KUKA KRL program: MyProgram_285().src

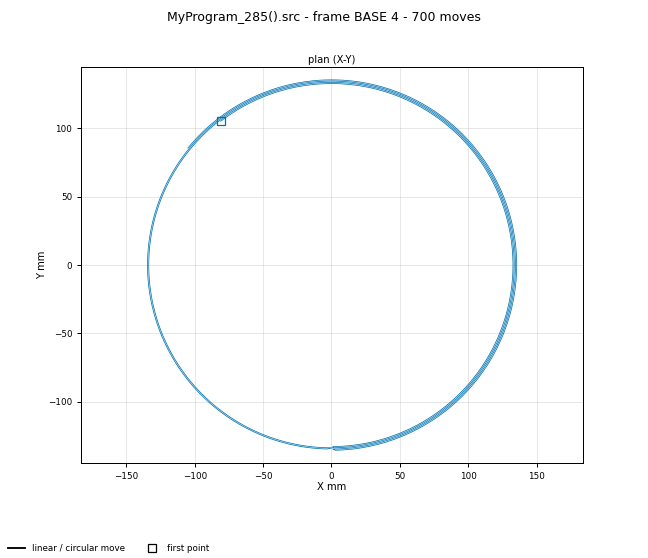
[picture p0: tool path of MyProgram_285().src in frame BASE 4, 700 of 700 moves have a stored position in this frame; points joined in program order, loops and branches not executed]
&ACCESS RVP
&REL 1
&PARAM TEMPLATE = C:\KRC\Roboter\Template\vorgabe
&PARAM EDITMASK = *
DEF MyProgram_285()
; ---- Setting reference (Base) ----
$BASE = BASE_DATA[4]

; --------------------------
; ---- Setting tool (TCP) ----
$TOOL = TOOL_DATA[3]
; --------------------------

$VEL.CP = VEL_APROX_PRINT
Startdeposition()
$VEL.CP = VEL_PRINT
LIN {X -81.057,Y 105.1926,Z 175,A 128.0118,B 7.901,C 0.1192,E1 7.8061,E2 323.7668} C_DIS
LIN {X -78.056,Y 107.4376,Z 175,A 126.422,B 7.9011,C 0.116,E1 7.8097,E2 325.352} C_DIS
LIN {X -74.6273,Y 109.8471,Z 175,A 124.5253,B 7.9011,C 0.1143,E1 7.8141,E2 327.2575} C_DIS
LIN {X -71.0281,Y 112.2079,Z 175,A 122.8509,B 7.9012,C 0.1087,E1 7.818,E2 328.9089} C_DIS
LIN {X -68.5302,Y 113.7507,Z 175,A 121.4995,B 7.9012,C 0.108,E1 7.8212,E2 330.2692} C_DIS
LIN {X -65.7271,Y 115.3929,Z 175,A 120.0866,B 7.9012,C 0.1062,E1 7.8246,E2 331.6823} C_DIS
LIN {X -62.604,Y 117.117,Z 175,A 118.509,B 7.9012,C 0.1046,E1 7.8285,E2 333.2631} C_DIS
LIN {X -59.7165,Y 118.6142,Z 175,A 117.111,B 7.9013,C 0.1027,E1 7.832,E2 334.6594} C_DIS
LIN {X -57.0613,Y 119.9128,Z 175,A 115.7895,B 7.9013,C 0.1017,E1 7.8353,E2 335.9852} C_DIS
LIN {X -53.8159,Y 121.4046,Z 175,A 114.2757,B 7.9013,C 0.0995,E1 7.8391,E2 337.4947} C_DIS
LIN {X -50.7871,Y 122.7025,Z 175,A 112.8825,B 7.9013,C 0.0974,E1 7.8427,E2 338.8834} C_DIS
LIN {X -48.0628,Y 123.7943,Z 175,A 111.5238,B 7.9013,C 0.0974,E1 7.8463,E2 340.252} C_DIS
LIN {X -44.7285,Y 125.0381,Z 175,A 110.0261,B 7.9013,C 0.0954,E1 7.8502,E2 341.7442} C_DIS
LIN {X -41.9571,Y 125.9947,Z 175,A 108.7023,B 7.9013,C 0.0951,E1 7.8537,E2 343.0739} C_DIS
LIN {X -38.5596,Y 127.0761,Z 175,A 107.2508,B 7.9014,C 0.0924,E1 7.8575,E2 344.5142} C_DIS
LIN {X -35.4154,Y 127.9882,Z 175,A 105.7886,B 7.9014,C 0.0921,E1 7.8615,E2 345.9813} C_DIS
LIN {X -32.266,Y 128.8183,Z 175,A 104.3779,B 7.9014,C 0.0911,E1 7.8653,E2 347.3918} C_DIS
LIN {X -29.4073,Y 129.5003,Z 175,A 103.0632,B 7.9014,C 0.0911,E1 7.8689,E2 348.711} C_DIS
LIN {X -25.8996,Y 130.2485,Z 175,A 101.5728,B 7.9014,C 0.0892,E1 7.873,E2 350.1939} C_DIS
LIN {X -22.6971,Y 130.8452,Z 175,A 100.1492,B 7.9014,C 0.0888,E1 7.8769,E2 351.6188} C_DIS
LIN {X -19.7973,Y 131.3144,Z 175,A 98.8772,B 7.9014,C 0.0883,E1 7.8804,E2 352.8906} C_DIS
LIN {X -16.5766,Y 131.7605,Z 175,A 97.4722,B 7.9014,C 0.0878,E1 7.8843,E2 354.2951} C_DIS
LIN {X -13.3289,Y 132.1284,Z 175,A 95.9474,B 7.9014,C 0.0892,E1 7.8885,E2 355.8326} C_DIS
LIN {X -9.1434,Y 132.4834,Z 175,A 94.0776,B 7.9014,C 0.0897,E1 7.8938,E2 357.7081} C_DIS
LIN {X -4.8868,Y 132.7079,Z 175,A 92.4029,B 7.9014,C 0.0868,E1 7.8984,E2 359.3627} C_DIS
LIN {X -2.3646,Y 132.7766,Z 175,A 91.2329,B 7.9014,C 0.088,E1 7.9017,E2 360.5417} C_DIS
LIN {X 1.6416,Y 132.7886,Z 175,A 89.665,B 7.9015,C 0.0854,E1 7.906,E2 362.09} C_DIS
LIN {X 4.5791,Y 132.7199,Z 175,A 88.2887,B 7.9015,C 0.0873,E1 7.9099,E2 363.4785} C_DIS
LIN {X 8.1447,Y 132.5475,Z 175,A 86.8344,B 7.9015,C 0.0861,E1 7.9139,E2 364.9221} C_DIS
LIN {X 11.3913,Y 132.3081,Z 175,A 85.3691,B 7.9015,C 0.0874,E1 7.918,E2 366.3939} C_DIS
LIN {X 14.6458,Y 131.988,Z 175,A 83.9666,B 7.9015,C 0.0877,E1 7.9219,E2 367.795} C_DIS
LIN {X 17.8755,Y 131.5902,Z 175,A 82.5679,B 7.9015,C 0.0881,E1 7.9258,E2 369.1926} C_DIS
LIN {X 21.0982,Y 131.1128,Z 175,A 81.1716,B 7.9015,C 0.0886,E1 7.9296,E2 370.5874} C_DIS
LIN {X 23.9902,Y 130.6138,Z 175,A 79.8272,B 7.9015,C 0.0905,E1 7.9333,E2 371.9406} C_DIS
LIN {X 26.9638,Y 130.0319,Z 175,A 78.5808,B 7.9015,C 0.0902,E1 7.9367,E2 373.1795} C_DIS
LIN {X 30.1009,Y 129.3419,Z 175,A 77.1406,B 7.9015,C 0.092,E1 7.9407,E2 374.6258} C_DIS
LIN {X 33.626,Y 128.4708,Z 175,A 75.6538,B 7.9015,C 0.0918,E1 7.9447,E2 376.1029} C_DIS
LIN {X 36.7252,Y 127.6194,Z 175,A 74.2858,B 7.9015,C 0.0925,E1 7.9483,E2 377.4684} C_DIS
LIN {X 39.8173,Y 126.6887,Z 175,A 72.9574,B 7.9015,C 0.0925,E1 7.9519,E2 378.7889} C_DIS
LIN {X 42.6193,Y 125.7742,Z 175,A 71.5511,B 7.9014,C 0.096,E1 7.9556,E2 380.2108} C_DIS
LIN {X 45.9756,Y 124.5862,Z 175,A 70.0956,B 7.9014,C 0.0961,E1 7.9594,E2 381.6566} C_DIS
LIN {X 49.3079,Y 123.3041,Z 175,A 68.4189,B 7.9014,C 0.1001,E1 7.9638,E2 383.3491} C_DIS
LIN {X 53.5228,Y 121.5357,Z 175,A 66.6106,B 7.9014,C 0.0995,E1 7.9684,E2 385.1382} C_DIS
LIN {X 56.7758,Y 120.0492,Z 175,A 65.0797,B 7.9014,C 0.1011,E1 7.9723,E2 386.6674} C_DIS
LIN {X 59.4163,Y 118.7657,Z 175,A 63.8092,B 7.9013,C 0.1028,E1 7.9755,E2 387.9384} C_DIS
LIN {X 62.2912,Y 117.2826,Z 175,A 62.4471,B 7.9013,C 0.104,E1 7.9788,E2 389.2965} C_DIS
LIN {X 65.4648,Y 115.5425,Z 175,A 60.8866,B 7.9013,C 0.1062,E1 7.9826,E2 390.857} C_DIS
LIN {X 68.2745,Y 113.9046,Z 175,A 59.4911,B 7.9013,C 0.1081,E1 7.986,E2 392.2517} C_DIS
LIN {X 71.0472,Y 112.1958,Z 175,A 58.1656,B 7.9013,C 0.1088,E1 7.9891,E2 393.5678} C_DIS
LIN {X 73.8328,Y 110.3825,Z 175,A 56.7558,B 7.9012,C 0.1106,E1 7.9924,E2 394.975} C_DIS
LIN {X 76.4862,Y 108.5607,Z 175,A 55.3298,B 7.9012,C 0.1136,E1 7.9957,E2 396.4055} C_DIS
LIN {X 79.2965,Y 106.5252,Z 175,A 53.7292,B 7.9011,C 0.118,E1 7.9993,E2 398.0185} C_DIS
LIN {X 82.472,Y 104.0866,Z 175,A 51.9965,B 7.9011,C 0.1211,E1 8.0031,E2 399.7522} C_DIS
LIN {X 86.0007,Y 101.1901,Z 175,A 50.1762,B 7.9011,C 0.122,E1 8.007,E2 401.5553} C_DIS
LIN {X 88.6934,Y 98.8385,Z 175,A 48.5255,B 7.901,C 0.1269,E1 8.0105,E2 403.2191} C_DIS
LIN {X 91.688,Y 96.067,Z 175,A 46.8002,B 7.901,C 0.1297,E1 8.014,E2 404.9407} C_DIS
LIN {X 94.4766,Y 93.3267,Z 175,A 45.1121,B 7.9008,C 0.1331,E1 8.0173,E2 406.6295} C_DIS
LIN {X 97.2976,Y 90.3812,Z 175,A 43.3866,B 7.9008,C 0.1362,E1 8.0206,E2 408.3515} C_DIS
LIN {X 100.3288,Y 87.005,Z 175,A 41.4834,B 7.9008,C 0.1394,E1 8.0241,E2 410.249} C_DIS
LIN {X 103.1083,Y 83.6923,Z 175,A 39.6732,B 7.9007,C 0.1424,E1 8.0273,E2 412.0533} C_DIS
LIN {X 105.6939,Y 80.402,Z 175,A 37.8145,B 7.9006,C 0.1475,E1 8.0305,E2 413.9191} C_DIS
LIN {X 108.3965,Y 76.719,Z 175,A 36.0259,B 7.9006,C 0.1487,E1 8.0334,E2 415.6868} C_DIS
LIN {X 110.4199,Y 73.7768,Z 175,A 34.5869,B 7.9006,C 0.1504,E1 8.0357,E2 417.1144} C_DIS
LIN {X 112.1939,Y 71.0502,Z 175,A 33.1857,B 7.9005,C 0.1537,E1 8.0378,E2 418.5161} C_DIS
LIN {X 113.7385,Y 68.5504,Z 175,A 31.8714,B 7.9004,C 0.1577,E1 8.0397,E2 419.8366} C_DIS
LIN {X 115.3839,Y 65.743,Z 175,A 30.4918,B 7.9004,C 0.1607,E1 8.0416,E2 421.2139} C_DIS
LIN {X 116.892,Y 63.0228,Z 175,A 29.1014,B 7.9003,C 0.165,E1 8.0435,E2 422.6109} C_DIS
LIN {X 118.621,Y 59.7031,Z 175,A 27.5765,B 7.9003,C 0.1674,E1 8.0454,E2 424.1259} C_DIS
LIN {X 119.9118,Y 57.0633,Z 175,A 26.294,B 7.9001,C 0.171,E1 8.047,E2 425.4109} C_DIS
LIN {X 121.4046,Y 53.816,Z 175,A 24.8414,B 7.9001,C 0.1733,E1 8.0486,E2 426.8538} C_DIS
LIN {X 122.69,Y 50.817,Z 175,A 23.474,B 7.9001,C 0.1762,E1 8.0501,E2 428.2172} C_DIS
LIN {X 123.7957,Y 48.0592,Z 175,A 22.1294,B 7.8999,C 0.1809,E1 8.0515,E2 429.5701} C_DIS
LIN {X 125.0375,Y 44.7301,Z 175,A 20.6688,B 7.8999,C 0.1836,E1 8.0529,E2 431.0231} C_DIS
LIN {X 125.9926,Y 41.9634,Z 175,A 19.3778,B 7.8998,C 0.1876,E1 8.0541,E2 432.3183} C_DIS
LIN {X 127.0728,Y 38.5704,Z 175,A 17.9165,B 7.8997,C 0.1903,E1 8.0553,E2 433.7717} C_DIS
LIN {X 127.9869,Y 35.42,Z 175,A 16.5296,B 7.8997,C 0.1937,E1 8.0563,E2 435.1562} C_DIS
LIN {X 128.9915,Y 31.5674,Z 175,A 14.7123,B 7.8994,C 0.2004,E1 8.0576,E2 436.9867} C_DIS
LIN {X 129.9196,Y 27.5006,Z 175,A 13.0796,B 7.8994,C 0.2022,E1 8.0585,E2 438.6008} C_DIS
LIN {X 130.4956,Y 24.6193,Z 175,A 11.8054,B 7.8993,C 0.2059,E1 8.0592,E2 439.8767} C_DIS
LIN {X 131.1125,Y 21.1001,Z 175,A 10.3294,B 7.8993,C 0.209,E1 8.0599,E2 441.346} C_DIS
LIN {X 131.5493,Y 18.1741,Z 175,A 9.074,B 7.8991,C 0.2122,E1 8.0604,E2 442.5999} C_DIS
LIN {X 131.9557,Y 14.946,Z 175,A 7.6671,B 7.8991,C 0.2163,E1 8.0609,E2 444.0084} C_DIS
LIN {X 132.2812,Y 11.7097,Z 175,A 6.293,B 7.8989,C 0.2198,E1 8.0612,E2 445.3801} C_DIS
LIN {X 132.5473,Y 8.1469,Z 175,A 4.8565,B 7.8989,C 0.2221,E1 8.0615,E2 446.8052} C_DIS
LIN {X 132.7082,Y 4.8784,Z 175,A 3.4177,B 7.8987,C 0.2267,E1 8.0617,E2 448.2485} C_DIS
LIN {X 132.7889,Y 1.6239,Z 175,A 2.0871,B 7.8987,C 0.2293,E1 8.0617,E2 449.5714} C_DIS
LIN {X 132.7888,Y -1.6303,Z 175,A 0.737,B 7.8986,C 0.2323,E1 8.0617,E2 450.9162} C_DIS
LIN {X 132.7204,Y -4.5652,Z 175,A -0.6124,B 7.8984,C 0.2376,E1 8.0617,E2 452.2767} C_DIS
LIN {X 132.5471,Y -8.1504,Z 175,A -2.0507,B 7.8984,C 0.2399,E1 8.0614,E2 453.7031} C_DIS
LIN {X 132.3075,Y -11.3988,Z 175,A -3.4885,B 7.8982,C 0.2446,E1 8.0611,E2 455.146} C_DIS
LIN {X 131.9888,Y -14.6388,Z 175,A -4.8638,B 7.8981,C 0.2481,E1 8.0607,E2 456.5191} C_DIS
LIN {X 131.5911,Y -17.8694,Z 175,A -6.2404,B 7.898,C 0.2515,E1 8.0602,E2 457.8937} C_DIS
LIN {X 131.1149,Y -21.0857,Z 175,A -7.6168,B 7.8979,C 0.255,E1 8.0596,E2 459.2682} C_DIS
LIN {X 130.612,Y -23.9998,Z 175,A -8.9463,B 7.8977,C 0.2597,E1 8.059,E2 460.6054} C_DIS
LIN {X 129.985,Y -27.1945,Z 175,A -10.2537,B 7.8977,C 0.2618,E1 8.0583,E2 461.9024} C_DIS
LIN {X 129.1722,Y -30.8178,Z 175,A -11.7399,B 7.8976,C 0.2641,E1 8.0573,E2 463.3759} C_DIS
LIN {X 128.47,Y -33.6291,Z 175,A -13.0564,B 7.8974,C 0.2689,E1 8.0564,E2 464.7018} C_DIS
LIN {X 127.6217,Y -36.7174,Z 175,A -14.3483,B 7.8974,C 0.271,E1 8.0555,E2 465.9841} C_DIS
LIN {X 126.7745,Y -39.545,Z 175,A -15.7264,B 7.8972,C 0.2766,E1 8.0543,E2 467.3762} C_DIS
LIN {X 125.5716,Y -43.2079,Z 175,A -17.2032,B 7.8972,C 0.2775,E1 8.053,E2 468.8318} C_DIS
LIN {X 124.5852,Y -45.9783,Z 175,A -18.5498,B 7.8969,C 0.2825,E1 8.0517,E2 470.1892} C_DIS
LIN {X 123.3033,Y -49.3099,Z 175,A -20.0641,B 7.8969,C 0.2862,E1 8.0502,E2 471.7019} C_DIS
LIN {X 122.1832,Y -52.0273,Z 175,A -21.3355,B 7.8967,C 0.2897,E1 8.0488,E2 472.975} C_DIS
LIN {X 120.8438,Y -55.0668,Z 175,A -22.805,B 7.8965,C 0.2942,E1 8.0471,E2 474.4503} C_DIS
LIN {X 119.3338,Y -58.2646,Z 175,A -24.1175,B 7.8965,C 0.2942,E1 8.0456,E2 475.7383} C_DIS
LIN {X 118.0208,Y -60.882,Z 175,A -25.4711,B 7.8963,C 0.2992,E1 8.0439,E2 477.1042} C_DIS
LIN {X 116.5021,Y -63.7406,Z 175,A -26.8694,B 7.8962,C 0.3028,E1 8.042,E2 478.5041} C_DIS
LIN {X 114.7343,Y -66.8712,Z 175,A -28.3677,B 7.8961,C 0.3057,E1 8.0399,E2 479.9975} C_DIS
LIN {X 113.0613,Y -69.6618,Z 175,A -29.7474,B 7.896,C 0.3088,E1 8.0379,E2 481.3757} C_DIS
LIN {X 110.9536,Y -72.9717,Z 175,A -31.531,B 7.8957,C 0.3148,E1 8.0352,E2 483.172} C_DIS
LIN {X 108.7302,Y -76.246,Z 175,A -33.154,B 7.8957,C 0.3173,E1 8.0327,E2 484.7864} C_DIS
LIN {X 106.4786,Y -79.3592,Z 175,A -34.8083,B 7.8955,C 0.3212,E1 8.0299,E2 486.4419} C_DIS
LIN {X 104.0884,Y -82.4698,Z 175,A -36.516,B 7.8953,C 0.3254,E1 8.027,E2 488.1531} C_DIS
LIN {X 101.2892,Y -85.8841,Z 175,A -38.3559,B 7.8952,C 0.3285,E1 8.0237,E2 489.9869} C_DIS
LIN {X 98.4102,Y -89.1684,Z 175,A -40.2454,B 7.895,C 0.3328,E1 8.0202,E2 491.8789} C_DIS
LIN {X 95.6134,Y -92.1614,Z 175,A -41.9873,B 7.8949,C 0.3361,E1 8.0168,E2 493.6194} C_DIS
LIN {X 92.6325,Y -95.1573,Z 175,A -43.7993,B 7.8947,C 0.3397,E1 8.0132,E2 495.4317} C_DIS
LIN {X 89.2595,Y -98.3276,Z 175,A -45.6603,B 7.8947,C 0.3412,E1 8.0095,E2 497.278} C_DIS
LIN {X 86.2402,Y -100.9865,Z 175,A -47.3866,B 7.8945,C 0.3445,E1 8.0058,E2 499.0047} C_DIS
LIN {X 83.0764,Y -103.6051,Z 175,A -49.1273,B 7.8944,C 0.3473,E1 8.0021,E2 500.7432} C_DIS
LIN {X 79.8864,Y -106.0837,Z 175,A -50.9481,B 7.8942,C 0.3519,E1 7.998,E2 502.5751} C_DIS
LIN {X 77.0562,Y -108.1571,Z 175,A -52.3961,B 7.8942,C 0.3534,E1 7.9947,E2 504.0164} C_DIS
LIN {X 73.779,Y -110.4184,Z 175,A -53.9372,B 7.8942,C 0.3531,E1 7.9912,E2 505.5373} C_DIS
LIN {X 71.0414,Y -112.1995,Z 175,A -55.3489,B 7.894,C 0.3554,E1 7.9879,E2 506.9507} C_DIS
LIN {X 68.4099,Y -113.8235,Z 175,A -56.7339,B 7.8939,C 0.3585,E1 7.9846,E2 508.343} C_DIS
LIN {X 65.6764,Y -115.4219,Z 175,A -58.0854,B 7.8938,C 0.3604,E1 7.9813,E2 509.6939} C_DIS
LIN {X 62.5927,Y -117.123,Z 175,A -59.6159,B 7.8937,C 0.3628,E1 7.9775,E2 511.227} C_DIS
LIN {X 59.6974,Y -118.6239,Z 175,A -60.9939,B 7.8937,C 0.3643,E1 7.9741,E2 512.6025} C_DIS
LIN {X 57.0567,Y -119.915,Z 175,A -62.286,B 7.8935,C 0.3664,E1 7.9709,E2 513.8986} C_DIS
LIN {X 53.8116,Y -121.4065,Z 175,A -63.7758,B 7.8935,C 0.3675,E1 7.9671,E2 515.3834} C_DIS
LIN {X 51.037,Y -122.5981,Z 175,A -65.0522,B 7.8935,C 0.3686,E1 7.9638,E2 516.6574} C_DIS
LIN {X 48.0932,Y -123.7824,Z 175,A -66.474,B 7.8933,C 0.3712,E1 7.9601,E2 518.0869} C_DIS
LIN {X 44.7465,Y -125.0316,Z 175,A -67.9549,B 7.8933,C 0.3718,E1 7.9562,E2 519.5614} C_DIS
LIN {X 41.9707,Y -125.9902,Z 175,A -69.2652,B 7.8932,C 0.3739,E1 7.9527,E2 520.878} C_DIS
LIN {X 38.5396,Y -127.0822,Z 175,A -70.7555,B 7.8932,C 0.3742,E1 7.9488,E2 522.3616} C_DIS
LIN {X 35.4139,Y -127.9886,Z 175,A -72.151,B 7.8932,C 0.3754,E1 7.945,E2 523.757} C_DIS
LIN {X 32.2635,Y -128.819,Z 175,A -73.5474,B 7.8931,C 0.3764,E1 7.9413,E2 525.1533} C_DIS
LIN {X 29.4043,Y -129.501,Z 175,A -74.8485,B 7.893,C 0.3779,E1 7.9377,E2 526.4592} C_DIS
LIN {X 25.8906,Y -130.2503,Z 175,A -76.3311,B 7.893,C 0.3779,E1 7.9337,E2 527.9346} C_DIS
LIN {X 22.6896,Y -130.8465,Z 175,A -77.7437,B 7.893,C 0.3788,E1 7.9298,E2 529.3491} C_DIS
LIN {X 19.791,Y -131.3154,Z 175,A -79.0064,B 7.893,C 0.3795,E1 7.9263,E2 530.612} C_DIS
LIN {X 16.8654,Y -131.7226,Z 175,A -80.3034,B 7.8929,C 0.3805,E1 7.9227,E2 531.9125} C_DIS
LIN {X 13.6246,Y -132.0979,Z 175,A -81.7555,B 7.8928,C 0.3819,E1 7.9187,E2 533.3709} C_DIS
LIN {X 10.0824,Y -132.4148,Z 175,A -83.2994,B 7.8928,C 0.3826,E1 7.9144,E2 534.9168} C_DIS
LIN {X 6.8219,Y -132.6222,Z 175,A -84.6801,B 7.8928,C 0.3826,E1 7.9105,E2 536.2947} C_DIS
LIN {X 3.2553,Y -132.7583,Z 175,A -86.149,B 7.8928,C 0.3816,E1 7.9064,E2 537.7556} C_DIS
LIN {X 0.9619,Y -132.7934,Z 175,A -86.8619,B 7.893,C 0.3771,E1 7.9045,E2 538.4349} C_DIS
Enddeposition()
LIN {X 0.9619,Y -132.7934,Z 175,A -86.8619,B 7.893,C 0.3771,E1 7.9045,E2 538.4349} C_DIS
Startdeposition()
$VEL.CP = VEL_PRINT
LIN {X 1.5089,Y -133.6974,Z 175,A -86.1199,B 7.8928,C 0.3729,E1 7.9063,E2 537.663} C_DIS
LIN {X 5.3626,Y -133.5965,Z 175,A -84.7785,B 7.8925,C 0.3779,E1 7.9099,E2 536.3596} C_DIS
LIN {X 8.2096,Y -133.4517,Z 175,A -83.4338,B 7.8927,C 0.3754,E1 7.9137,E2 534.999} C_DIS
LIN {X 10.8852,Y -133.2606,Z 175,A -82.3895,B 7.8926,C 0.3769,E1 7.9166,E2 533.9671} C_DIS
LIN {X 14.074,Y -132.9613,Z 175,A -81.0844,B 7.8926,C 0.3775,E1 7.9202,E2 532.6697} C_DIS
LIN {X 16.6031,Y -132.6712,Z 175,A -79.6231,B 7.8929,C 0.3705,E1 7.9243,E2 531.1615} C_DIS
LIN {X 20.8494,Y -132.0688,Z 175,A -77.9423,B 7.8929,C 0.3723,E1 7.9289,E2 529.4993} C_DIS
LIN {X 24.3534,Y -131.4692,Z 175,A -76.3074,B 7.8929,C 0.3693,E1 7.9335,E2 527.8494} C_DIS
LIN {X 27.7753,Y -130.7877,Z 175,A -74.8789,B 7.8929,C 0.3695,E1 7.9374,E2 526.4283} C_DIS
LIN {X 30.8025,Y -130.1083,Z 175,A -73.5664,B 7.8929,C 0.3687,E1 7.9409,E2 525.1171} C_DIS
LIN {X 34.5915,Y -129.1515,Z 175,A -71.9151,B 7.893,C 0.3677,E1 7.9454,E2 523.4676} C_DIS
LIN {X 38.6164,Y -128.0067,Z 175,A -70.1119,B 7.8931,C 0.3659,E1 7.9502,E2 521.6619} C_DIS
LIN {X 42.2857,Y -126.8407,Z 175,A -68.521,B 7.8931,C 0.3653,E1 7.9544,E2 520.0772} C_DIS
LIN {X 45.9701,Y -125.5541,Z 175,A -66.8639,B 7.8932,C 0.3638,E1 7.9588,E2 518.4207} C_DIS
LIN {X 49.6498,Y -124.1437,Z 175,A -65.1683,B 7.8932,C 0.3617,E1 7.9632,E2 516.723} C_DIS
LIN {X 52.3902,Y -123.0139,Z 175,A -63.8232,B 7.8934,C 0.3588,E1 7.9667,E2 515.3676} C_DIS
LIN {X 56.2576,Y -121.2919,Z 175,A -62.1294,B 7.8934,C 0.3586,E1 7.971,E2 513.6874} C_DIS
LIN {X 59.333,Y -119.8176,Z 175,A -60.5388,B 7.8936,C 0.3542,E1 7.975,E2 512.0794} C_DIS
LIN {X 62.807,Y -118.0357,Z 175,A -58.5941,B 7.894,C 0.3467,E1 7.9799,E2 510.0992} C_DIS
LIN {X 66.3498,Y -116.0813,Z 175,A -56.8538,B 7.894,C 0.3439,E1 7.9841,E2 508.3566} C_DIS
LIN {X 69.9288,Y -113.961,Z 175,A -55.4646,B 7.8939,C 0.3485,E1 7.9873,E2 507.0154} C_DIS
LIN {X 73.7335,Y -111.5374,Z 175,A -53.5154,B 7.894,C 0.345,E1 7.9919,E2 505.0625} C_DIS
LIN {X 76.8479,Y -109.4149,Z 175,A -51.8208,B 7.8942,C 0.3407,E1 7.9958,E2 503.3564} C_DIS
LIN {X 80.6231,Y -106.6634,Z 175,A -49.4886,B 7.8946,C 0.3307,E1 8.0011,E2 500.9808} C_DIS
LIN {X 84.3837,Y -103.7142,Z 175,A -47.9291,B 7.8944,C 0.3362,E1 8.0044,E2 499.4809} C_DIS
LIN {X 87.8026,Y -100.8359,Z 175,A -46.0622,B 7.8945,C 0.3334,E1 8.0083,E2 497.6183} C_DIS
LIN {X 90.9521,Y -98.0047,Z 175,A -44.2515,B 7.8947,C 0.3298,E1 8.012,E2 495.8064} C_DIS
LIN {X 94.1067,Y -94.9795,Z 175,A -42.4332,B 7.8948,C 0.327,E1 8.0157,E2 493.9932} C_DIS
LIN {X 96.9679,Y -92.0573,Z 175,A -40.6647,B 7.895,C 0.3229,E1 8.0191,E2 492.2211} C_DIS
LIN {X 99.9709,Y -88.7866,Z 175,A -38.987,B 7.895,C 0.3231,E1 8.0222,E2 490.5696} C_DIS
LIN {X 103.0647,Y -85.1753,Z 175,A -36.8649,B 7.8952,C 0.3168,E1 8.026,E2 488.435} C_DIS
LIN {X 105.9684,Y -81.5352,Z 175,A -34.7551,B 7.8955,C 0.3099,E1 8.0297,E2 486.309} C_DIS
LIN {X 109.1799,Y -77.1811,Z 175,A -32.3222,B 7.8958,C 0.3021,E1 8.0337,E2 483.8594} C_DIS
LIN {X 111.1292,Y -74.347,Z 175,A -31.1607,B 7.8957,C 0.3046,E1 8.0355,E2 482.7355} C_DIS
LIN {X 112.8664,Y -71.6829,Z 175,A -29.736,B 7.8959,C 0.3,E1 8.0376,E2 481.3018} C_DIS
LIN {X 114.7538,Y -68.6204,Z 175,A -28.2325,B 7.8959,C 0.2969,E1 8.0398,E2 479.8015} C_DIS
LIN {X 118.0174,Y -62.8418,Z 175,A -25.4849,B 7.8962,C 0.2915,E1 8.0435,E2 477.0631} C_DIS
LIN {X 119.4816,Y -60.0107,Z 175,A -23.7349,B 7.8966,C 0.2803,E1 8.0457,E2 475.2637} C_DIS
LIN {X 121.2483,Y -56.3518,Z 175,A -22.0037,B 7.8967,C 0.2758,E1 8.0478,E2 473.532} C_DIS
LIN {X 123.0433,Y -52.3221,Z 175,A -20.4528,B 7.8967,C 0.2776,E1 8.0494,E2 472.0217} C_DIS
LIN {X 124.654,Y -48.353,Z 175,A -18.8899,B 7.8967,C 0.278,E1 8.051,E2 470.4909} C_DIS
LIN {X 125.6151,Y -45.8008,Z 175,A -17.6349,B 7.8968,C 0.2731,E1 8.0522,E2 469.224} C_DIS
LIN {X 126.5099,Y -43.2688,Z 175,A -16.2571,B 7.8971,C 0.2654,E1 8.0535,E2 467.8168} C_DIS
LIN {X 127.5151,Y -40.2093,Z 175,A -15.1252,B 7.8971,C 0.2665,E1 8.0544,E2 466.7146} C_DIS
LIN {X 129.5325,Y -33.1371,Z 175,A -11.6828,B 7.8975,C 0.2519,E1 8.057,E2 463.2329} C_DIS
LIN {X 130.4529,Y -29.3077,Z 175,A -10.4412,B 7.8975,C 0.2561,E1 8.0577,E2 462.0452} C_DIS
LIN {X 131.281,Y -25.3388,Z 175,A -8.6465,B 7.8975,C 0.25,E1 8.0587,E2 460.2417} C_DIS
LIN {X 132.0441,Y -21.0087,Z 175,A -6.778,B 7.8978,C 0.2449,E1 8.0596,E2 458.3734} C_DIS
LIN {X 132.5387,Y -17.6145,Z 175,A -5.5257,B 7.8978,C 0.245,E1 8.0601,E2 457.1466} C_DIS
LIN {X 132.9231,Y -14.4285,Z 175,A -4.0577,B 7.8979,C 0.2392,E1 8.0605,E2 455.6658} C_DIS
LIN {X 133.2729,Y -10.74,Z 175,A -2.4359,B 7.8981,C 0.234,E1 8.0609,E2 454.0384} C_DIS
LIN {X 133.5589,Y -6.2439,Z 175,A -0.536,B 7.8982,C 0.229,E1 8.0612,E2 452.1406} C_DIS
LIN {X 133.6764,Y -2.7732,Z 175,A 0.9477,B 7.8983,C 0.2248,E1 8.0613,E2 450.6561} C_DIS
LIN {X 133.7022,Y 0.8628,Z 175,A 2.4681,B 7.8985,C 0.2211,E1 8.0613,E2 449.139} C_DIS
LIN {X 133.5823,Y 5.7262,Z 175,A 4.5294,B 7.8986,C 0.2155,E1 8.0611,E2 447.0788} C_DIS
LIN {X 133.3258,Y 10.0537,Z 175,A 6.2079,B 7.8986,C 0.2138,E1 8.0608,E2 445.4208} C_DIS
LIN {X 132.9649,Y 14.0404,Z 175,A 7.8868,B 7.8988,C 0.2096,E1 8.0604,E2 443.745} C_DIS
LIN {X 132.6373,Y 16.8618,Z 175,A 9.1313,B 7.8988,C 0.2055,E1 8.0599,E2 442.4961} C_DIS
LIN {X 132.162,Y 20.2477,Z 175,A 10.4996,B 7.8989,C 0.2033,E1 8.0594,E2 441.1385} C_DIS
LIN {X 131.6978,Y 23.0788,Z 175,A 11.7566,B 7.899,C 0.1993,E1 8.0588,E2 439.8771} C_DIS
LIN {X 131.1891,Y 25.8192,Z 175,A 13.035,B 7.8992,C 0.1942,E1 8.0581,E2 438.5876} C_DIS
LIN {X 130.5026,Y 29.0902,Z 175,A 14.3844,B 7.8992,C 0.1918,E1 8.0573,E2 437.2473} C_DIS
LIN {X 129.6523,Y 32.6652,Z 175,A 15.8978,B 7.8992,C 0.1887,E1 8.0563,E2 435.7402} C_DIS
LIN {X 128.8081,Y 35.8493,Z 175,A 17.2033,B 7.8993,C 0.1868,E1 8.0554,E2 434.4466} C_DIS
LIN {X 127.9896,Y 38.6723,Z 175,A 18.9574,B 7.8996,C 0.1736,E1 8.0539,E2 432.631} C_DIS
LIN {X 126.7465,Y 42.5686,Z 175,A 20.2913,B 7.8996,C 0.1771,E1 8.0528,E2 431.3473} C_DIS
LIN {X 124.1627,Y 49.6026,Z 175,A 23.2242,B 7.8996,C 0.174,E1 8.0499,E2 428.4464} C_DIS
LIN {X 122.9236,Y 52.5992,Z 175,A 24.8032,B 7.8998,C 0.1666,E1 8.0482,E2 426.8434} C_DIS
LIN {X 121.4678,Y 55.8771,Z 175,A 26.1812,B 7.8998,C 0.1657,E1 8.0466,E2 425.4839} C_DIS
LIN {X 120.2411,Y 58.4745,Z 175,A 27.6616,B 7.9,C 0.1576,E1 8.0448,E2 423.9723} C_DIS
LIN {X 118.3614,Y 62.1867,Z 175,A 29.1889,B 7.9,C 0.1581,E1 8.0429,E2 422.4753} C_DIS
LIN {X 116.3547,Y 65.8704,Z 175,A 31.1294,B 7.9,C 0.1508,E1 8.0402,E2 420.5165} C_DIS
LIN {X 114.1728,Y 69.5836,Z 175,A 32.9359,B 7.9002,C 0.147,E1 8.0376,E2 418.7138} C_DIS
LIN {X 111.9848,Y 73.0522,Z 175,A 34.6429,B 7.9002,C 0.1438,E1 8.0351,E2 417.012} C_DIS
LIN {X 109.6985,Y 76.4421,Z 175,A 36.2105,B 7.9002,C 0.1432,E1 8.0326,E2 415.4661} C_DIS
LIN {X 107.0104,Y 80.1627,Z 175,A 39.4666,B 7.9007,C 0.1137,E1 8.0269,E2 412.0508} C_DIS
LIN {X 101.7687,Y 86.7197,Z 175,A 41.7708,B 7.9005,C 0.1307,E1 8.0231,E2 409.9043} C_DIS
LIN {X 99.1513,Y 89.7006,Z 175,A 43.5285,B 7.9005,C 0.126,E1 8.0198,E2 408.1389} C_DIS
LIN {X 96.3018,Y 92.7536,Z 175,A 45.3138,B 7.9005,C 0.1224,E1 8.0163,E2 406.3535} C_DIS
LIN {X 94.0145,Y 95.0711,Z 175,A 46.6717,B 7.9006,C 0.1203,E1 8.0137,E2 404.9998} C_DIS
LIN {X 90.7682,Y 98.1755,Z 175,A 48.5977,B 7.9006,C 0.1165,E1 8.0097,E2 403.0731} C_DIS
LIN {X 87.3827,Y 101.2,Z 175,A 50.4912,B 7.9007,C 0.1138,E1 8.0058,E2 401.1854} C_DIS
LIN {X 83.8748,Y 104.1257,Z 175,A 52.3805,B 7.9007,C 0.1115,E1 8.0017,E2 399.3041} C_DIS
LIN {X 80.7106,Y 106.5974,Z 175,A 54.1754,B 7.9008,C 0.1071,E1 7.9977,E2 397.4998} C_DIS
LIN {X 78.2136,Y 108.4429,Z 175,A 56.2447,B 7.901,C 0.0912,E1 7.9928,E2 395.3404} C_DIS
LIN {X 72.9024,Y 112.0821,Z 175,A 58.2016,B 7.9009,C 0.1017,E1 7.9885,E2 393.481} C_DIS
LIN {X 68.9848,Y 114.5351,Z 175,A 60.1293,B 7.9009,C 0.0997,E1 7.9839,E2 391.5596} C_DIS
LIN {X 65.2744,Y 116.6897,Z 175,A 61.9628,B 7.9009,C 0.0972,E1 7.9795,E2 389.7267} C_DIS
LIN {X 61.3166,Y 118.8168,Z 175,A 63.9246,B 7.9009,C 0.0939,E1 7.9746,E2 387.7605} C_DIS
LIN {X 57.7242,Y 120.6007,Z 175,A 65.272,B 7.9009,C 0.0984,E1 7.9713,E2 386.4576} C_DIS
LIN {X 55.2243,Y 121.7677,Z 175,A 66.6508,B 7.9009,C 0.0935,E1 7.9678,E2 385.0554} C_DIS
LIN {X 51.7537,Y 123.2811,Z 175,A 68.2577,B 7.9009,C 0.092,E1 7.9636,E2 383.4504} C_DIS
LIN {X 48.5452,Y 124.5793,Z 175,A 69.7687,B 7.901,C 0.0899,E1 7.9597,E2 381.9362} C_DIS
LIN {X 44.7125,Y 126.0075,Z 175,A 71.7972,B 7.901,C 0.0833,E1 7.9543,E2 379.8748} C_DIS
LIN {X 41.4457,Y 127.1202,Z 175,A 72.9255,B 7.901,C 0.0882,E1 7.9514,E2 378.7889} C_DIS
LIN {X 35.9742,Y 128.7731,Z 175,A 75.7904,B 7.9011,C 0.079,E1 7.9436,E2 375.8745} C_DIS
LIN {X 32.1015,Y 129.7952,Z 175,A 77.2527,B 7.9011,C 0.0822,E1 7.9397,E2 374.4433} C_DIS
LIN {X 28.7713,Y 130.5727,Z 175,A 78.5858,B 7.9011,C 0.0836,E1 7.9361,E2 373.1265} C_DIS
LIN {X 25.5689,Y 131.237,Z 175,A 80.0137,B 7.9011,C 0.0823,E1 7.9322,E2 371.6957} C_DIS
LIN {X 22.1742,Y 131.8523,Z 175,A 81.4866,B 7.9011,C 0.0817,E1 7.9282,E2 370.2239} C_DIS
LIN {X 18.4516,Y 132.4253,Z 175,A 83.1232,B 7.9011,C 0.0807,E1 7.9236,E2 368.5851} C_DIS
LIN {X 14.6735,Y 132.8968,Z 175,A 84.4753,B 7.9011,C 0.0848,E1 7.92,E2 367.2671} C_DIS
LIN {X 11.4787,Y 133.2105,Z 175,A 86.0842,B 7.9011,C 0.0806,E1 7.9154,E2 365.6308} C_DIS
LIN {X 7.2097,Y 133.5104,Z 175,A 87.8607,B 7.9011,C 0.0812,E1 7.9105,E2 363.8619} C_DIS
LIN {X 4.2983,Y 133.6362,Z 175,A 89.2496,B 7.9011,C 0.0788,E1 7.9066,E2 362.4568} C_DIS
LIN {X 0.7245,Y 133.7021,Z 175,A 90.8263,B 7.9011,C 0.078,E1 7.9022,E2 360.8753} C_DIS
LIN {X -3.4331,Y 133.6602,Z 175,A 92.3315,B 7.9011,C 0.0826,E1 7.8981,E2 359.4041} C_DIS
LIN {X -6.3068,Y 133.5558,Z 175,A 93.7057,B 7.9011,C 0.0805,E1 7.8942,E2 358.0136} C_DIS
LIN {X -10.1733,Y 133.3171,Z 175,A 95.4501,B 7.9011,C 0.0794,E1 7.8893,E2 356.2599} C_DIS
LIN {X -14.4238,Y 132.9237,Z 175,A 97.1817,B 7.9011,C 0.0816,E1 7.8845,E2 354.5409} C_DIS
LIN {X -18.5381,Y 132.413,Z 175,A 98.8871,B 7.9011,C 0.0834,E1 7.8798,E2 352.8451} C_DIS
LIN {X -22.0263,Y 131.877,Z 175,A 100.4336,B 7.9011,C 0.0835,E1 7.8755,E2 351.2953} C_DIS
LIN {X -24.9449,Y 131.3563,Z 175,A 101.629,B 7.9011,C 0.0854,E1 7.8723,E2 350.1096} C_DIS
LIN {X -27.8485,Y 130.7719,Z 175,A 103.0617,B 7.9011,C 0.0836,E1 7.8683,E2 348.6582} C_DIS
LIN {X -31.8999,Y 129.8438,Z 175,A 104.8831,B 7.9011,C 0.0841,E1 7.8634,E2 346.8332} C_DIS
LIN {X -36.4981,Y 128.6266,Z 175,A 107.2052,B 7.9011,C 0.0813,E1 7.857,E2 344.4784} C_DIS
LIN {X -40.0133,Y 127.5777,Z 175,A 108.5457,B 7.9011,C 0.0862,E1 7.8535,E2 343.1668} C_DIS
LIN {X -43.9725,Y 126.266,Z 175,A 110.1929,B 7.9011,C 0.0901,E1 7.8492,E2 341.5375} C_DIS
LIN {X -47.8059,Y 124.8667,Z 175,A 112.5726,B 7.9011,C 0.0821,E1 7.8428,E2 339.0834} C_DIS
LIN {X -52.2817,Y 123.0606,Z 175,A 114.2102,B 7.9011,C 0.0911,E1 7.8387,E2 337.4992} C_DIS
LIN {X -55.6032,Y 121.5945,Z 175,A 115.5251,B 7.9009,C 0.0966,E1 7.8354,E2 336.2143} C_DIS
LIN {X -58.936,Y 120.0134,Z 175,A 117.3871,B 7.9009,C 0.0943,E1 7.8307,E2 334.3199} C_DIS
LIN {X -63.3856,Y 117.7261,Z 175,A 119.3119,B 7.9009,C 0.1005,E1 7.826,E2 332.4231} C_DIS
LIN {X -66.513,Y 115.9882,Z 175,A 121.0307,B 7.9009,C 0.1,E1 7.8218,E2 330.6834} C_DIS
LIN {X -70.4516,Y 113.6388,Z 175,A 122.7467,B 7.9009,C 0.1066,E1 7.8177,E2 328.9988} C_DIS
LIN {X -73.7209,Y 111.5457,Z 175,A 124.6491,B 7.9009,C 0.1057,E1 7.8132,E2 327.0694} C_DIS
LIN {X -77.1432,Y 109.2066,Z 175,A 126.4874,B 7.9008,C 0.1078,E1 7.809,E2 325.2251} C_DIS
LIN {X -80.1257,Y 107.038,Z 175,A 128.1085,B 7.9008,C 0.1099,E1 7.8053,E2 323.6005} C_DIS
LIN {X -83.4577,Y 104.4606,Z 175,A 129.8987,B 7.9008,C 0.1134,E1 7.8014,E2 321.8138} C_DIS
LIN {X -86.8351,Y 101.6706,Z 175,A 131.5934,B 7.9006,C 0.1195,E1 7.7978,E2 320.1426} C_DIS
LIN {X -89.3924,Y 99.4294,Z 175,A 133.2909,B 7.9006,C 0.1188,E1 7.7942,E2 318.4177} C_DIS
LIN {X -92.6778,Y 96.3749,Z 175,A 135.1285,B 7.9006,C 0.1239,E1 7.7905,E2 316.5921} C_DIS
LIN {X -95.2866,Y 93.7959,Z 175,A 136.8522,B 7.9006,C 0.125,E1 7.7871,E2 314.8516} C_DIS
LIN {X -98.6323,Y 90.2712,Z 175,A 138.8638,B 7.9005,C 0.1304,E1 7.7833,E2 312.8505} C_DIS
LIN {X -101.3351,Y 87.2258,Z 175,A 140.6825,B 7.9005,C 0.1332,E1 7.7799,E2 311.0246} C_DIS
LIN {X -104.2528,Y 83.7173,Z 175,A 142.6025,B 7.9003,C 0.1381,E1 7.7765,E2 309.1108} C_DIS
LIN {X -106.4225,Y 80.9414,Z 175,A 144.1881,B 7.9003,C 0.1405,E1 7.7738,E2 307.5176} C_DIS
LIN {X -109.1208,Y 77.2649,Z 175,A 146.8885,B 7.9003,C 0.1346,E1 7.7693,E2 304.7289} C_DIS
LIN {X -112.2884,Y 72.5846,Z 175,A 149.3946,B 7.9003,C 0.1393,E1 7.7655,E2 302.215} C_DIS
LIN {X -115.3686,Y 67.5815,Z 175,A 151.518,B 7.9001,C 0.1511,E1 7.7626,E2 300.1419} C_DIS
LIN {X -117.1629,Y 64.4206,Z 175,A 152.9096,B 7.9,C 0.1574,E1 7.7607,E2 298.7719} C_DIS
LIN {X -118.7868,Y 61.3755,Z 175,A 154.4018,B 7.8999,C 0.161,E1 7.7588,E2 297.2796} C_DIS
LIN {X -120.3961,Y 58.1525,Z 175,A 155.8167,B 7.8998,C 0.1668,E1 7.7571,E2 295.8817} C_DIS
LIN {X -121.6839,Y 55.4099,Z 175,A 157.2751,B 7.8998,C 0.168,E1 7.7554,E2 294.4054} C_DIS
LIN {X -123.0845,Y 52.2246,Z 175,A 158.6009,B 7.8996,C 0.1743,E1 7.7539,E2 293.101} C_DIS
LIN {X -124.7486,Y 48.1097,Z 175,A 160.7135,B 7.8996,C 0.1765,E1 7.7517,E2 290.9648} C_DIS
LIN {X -126.0185,Y 44.682,Z 175,A 162.2942,B 7.8995,C 0.1806,E1 7.7502,E2 289.3839} C_DIS
LIN {X -127.1962,Y 41.2077,Z 175,A 163.6693,B 7.8993,C 0.1876,E1 7.749,E2 288.0341} C_DIS
LIN {X -128.2925,Y 37.6524,Z 175,A 165.2638,B 7.8993,C 0.192,E1 7.7477,E2 286.4412} C_DIS
LIN {X -128.96,Y 35.3059,Z 175,A 166.6467,B 7.8993,C 0.1904,E1 7.7467,E2 285.0185} C_DIS
LIN {X -129.9791,Y 31.3386,Z 175,A 168.3026,B 7.8991,C 0.1966,E1 7.7456,E2 283.3763} C_DIS
LIN {X -130.9207,Y 27.1422,Z 175,A 170.1787,B 7.899,C 0.2014,E1 7.7445,E2 281.498} C_DIS
LIN {X -131.6306,Y 23.4542,Z 175,A 171.8747,B 7.8989,C 0.2048,E1 7.7436,E2 279.793} C_DIS
LIN {X -132.3104,Y 19.2562,Z 175,A 173.6558,B 7.8987,C 0.2106,E1 7.7429,E2 278.0186} C_DIS
LIN {X -132.73,Y 16.1102,Z 175,A 174.843,B 7.8986,C 0.2168,E1 7.7425,E2 276.8536} C_DIS
LIN {X -133.0508,Y 13.2057,Z 175,A 176.3471,B 7.8986,C 0.217,E1 7.742,E2 275.3202} C_DIS
LIN {X -133.3868,Y 9.218,Z 175,A 178.1065,B 7.8984,C 0.2213,E1 7.7416,E2 273.5569} C_DIS
LIN {X -133.5786,Y 5.8213,Z 175,A 179.5592,B 7.8984,C 0.2256,E1 7.7414,E2 272.1062} C_DIS
LIN {X -133.674,Y 2.92,Z 175,A -179.0431,B 7.8983,C 0.2271,E1 7.7414,E2 270.6909} C_DIS
LIN {X -133.6986,Y -1.389,Z 175,A -177.2109,B 7.8981,C 0.2326,E1 7.7414,E2 268.8621} C_DIS
LIN {X -133.5881,Y -5.5772,Z 175,A -175.4725,B 7.8979,C 0.2386,E1 7.7415,E2 267.1322} C_DIS
LIN {X -133.3395,Y -9.8658,Z 175,A -173.6363,B 7.8978,C 0.2439,E1 7.7419,E2 265.2981} C_DIS
LIN {X -132.9933,Y -13.7766,Z 175,A -171.7732,B 7.8978,C 0.2463,E1 7.7424,E2 263.4144} C_DIS
LIN {X -132.4708,Y -18.1329,Z 175,A -169.8633,B 7.8976,C 0.2513,E1 7.7431,E2 261.5024} C_DIS
LIN {X -131.8815,Y -21.9994,Z 175,A -168.4249,B 7.8973,C 0.2592,E1 7.7437,E2 260.0943} C_DIS
LIN {X -131.3548,Y -24.9525,Z 175,A -167.1848,B 7.8972,C 0.2635,E1 7.7443,E2 258.8607} C_DIS
LIN {X -130.5157,Y -29.0329,Z 175,A -165.1513,B 7.8972,C 0.2651,E1 7.7455,E2 256.7984} C_DIS
LIN {X -129.19,Y -34.4471,Z 175,A -162.5254,B 7.897,C 0.2685,E1 7.7473,E2 254.1452} C_DIS
LIN {X -127.7419,Y -39.4814,Z 175,A -160.3646,B 7.8967,C 0.2758,E1 7.749,E2 251.9963} C_DIS
LIN {X -126.6057,Y -42.9914,Z 175,A -158.6913,B 7.8967,C 0.2788,E1 7.7505,E2 250.3129} C_DIS
LIN {X -125.3905,Y -46.4125,Z 175,A -157.1889,B 7.8965,C 0.2837,E1 7.7519,E2 248.818} C_DIS
LIN {X -124.0858,Y -49.7934,Z 175,A -155.6625,B 7.8963,C 0.2882,E1 7.7535,E2 247.2958} C_DIS
LIN {X -122.8056,Y -52.8719,Z 175,A -154.2393,B 7.8962,C 0.292,E1 7.755,E2 245.8743} C_DIS
LIN {X -121.4839,Y -55.8423,Z 175,A -152.577,B 7.8962,C 0.2918,E1 7.757,E2 244.1797} C_DIS
LIN {X -119.3893,Y -60.192,Z 175,A -150.652,B 7.8959,C 0.2991,E1 7.7594,E2 242.2737} C_DIS
LIN {X -117.7374,Y -63.3645,Z 175,A -148.3653,B 7.8962,C 0.2922,E1 7.7625,E2 239.8945} C_DIS
LIN {X -114.9318,Y -68.3217,Z 175,A -146.5755,B 7.8956,C 0.3075,E1 7.7649,E2 238.1869} C_DIS
LIN {X -112.6242,Y -72.0621,Z 175,A -144.6711,B 7.8954,C 0.3117,E1 7.7678,E2 236.2807} C_DIS
LIN {X -110.0146,Y -75.9874,Z 175,A -142.6431,B 7.8952,C 0.3163,E1 7.7709,E2 234.2528} C_DIS
LIN {X -107.7428,Y -79.1747,Z 175,A -140.9593,B 7.8951,C 0.3201,E1 7.7737,E2 232.5689} C_DIS
LIN {X -105.4059,Y -82.2611,Z 175,A -139.0562,B 7.8951,C 0.3201,E1 7.777,E2 230.6363} C_DIS
LIN {X -102.2907,Y -86.1034,Z 175,A -137.0612,B 7.8948,C 0.3266,E1 7.7805,E2 228.6575} C_DIS
LIN {X -99.3044,Y -89.5319,Z 175,A -135.2028,B 7.8946,C 0.332,E1 7.7839,E2 226.811} C_DIS
LIN {X -96.174,Y -92.8856,Z 175,A -133.1081,B 7.8946,C 0.3341,E1 7.788,E2 224.701} C_DIS
LIN {X -93.658,Y -95.4218,Z 175,A -131.5517,B 7.8944,C 0.3367,E1 7.7911,E2 223.1418} C_DIS
LIN {X -89.1397,Y -99.6557,Z 175,A -128.877,B 7.8942,C 0.3414,E1 7.7966,E2 220.4652} C_DIS
LIN {X -85.7414,Y -102.5945,Z 175,A -126.923,B 7.8941,C 0.3444,E1 7.8007,E2 218.5081} C_DIS
LIN {X -82.051,Y -105.569,Z 175,A -124.9209,B 7.8939,C 0.3483,E1 7.8051,E2 216.51} C_DIS
LIN {X -78.9706,Y -107.8927,Z 175,A -122.8872,B 7.894,C 0.3451,E1 7.8098,E2 214.4292} C_DIS
LIN {X -75.9071,Y -110.0698,Z 175,A -121.5379,B 7.8937,C 0.3517,E1 7.8128,E2 213.1127} C_DIS
LIN {X -72.1962,Y -112.5383,Z 175,A -119.7202,B 7.8936,C 0.3559,E1 7.817,E2 211.3066} C_DIS
LIN {X -69.2942,Y -114.348,Z 175,A -118.1304,B 7.8936,C 0.3561,E1 7.8208,E2 209.7015} C_DIS
LIN {X -65.3174,Y -116.6655,Z 175,A -116.2218,B 7.8934,C 0.3597,E1 7.8255,E2 207.8008} C_DIS
LIN {X -61.9626,Y -118.4791,Z 175,A -114.6113,B 7.8933,C 0.3621,E1 7.8294,E2 206.1932} C_DIS
LIN {X -58.5056,Y -120.2257,Z 175,A -112.9333,B 7.8933,C 0.3638,E1 7.8336,E2 204.513} C_DIS
LIN {X -54.8791,Y -121.9221,Z 175,A -111.1334,B 7.8932,C 0.3643,E1 7.8382,E2 202.7025} C_DIS
LIN {X -51.1558,Y -123.5308,Z 175,A -109.3787,B 7.8932,C 0.3658,E1 7.8427,E2 200.9455} C_DIS
LIN {X -47.4669,Y -124.9956,Z 175,A -107.4804,B 7.8932,C 0.3642,E1 7.8477,E2 199.0224} C_DIS
LIN {X -43.9209,Y -126.2839,Z 175,A -105.4441,B 7.8934,C 0.3587,E1 7.8533,E2 196.9331} C_DIS
LIN {X -38.9326,Y -127.9099,Z 175,A -103.4527,B 7.8932,C 0.3646,E1 7.8585,E2 194.9736} C_DIS
LIN {X -35.1291,Y -129.0082,Z 175,A -101.9872,B 7.8929,C 0.3695,E1 7.8624,E2 193.5368} C_DIS
LIN {X -31.145,Y -130.0258,Z 175,A -100.3708,B 7.8928,C 0.3729,E1 7.8667,E2 191.9381} C_DIS
LIN {X -27.069,Y -130.9356,Z 175,A -98.561,B 7.8928,C 0.3735,E1 7.8716,E2 190.1254} C_DIS
LIN {X -23.6483,Y -131.5958,Z 175,A -97.1003,B 7.8927,C 0.3746,E1 7.8756,E2 188.6682} C_DIS
LIN {X -20.3456,Y -132.1468,Z 175,A -95.6206,B 7.8927,C 0.3744,E1 7.8797,E2 187.1825} C_DIS
LIN {X -16.5315,Y -132.6798,Z 175,A -93.7985,B 7.8928,C 0.3719,E1 7.8849,E2 185.3383} C_DIS
LIN {X -11.7023,Y -133.1916,Z 175,A -91.8803,B 7.8927,C 0.375,E1 7.8901,E2 183.4397} C_DIS
LIN {X -7.7524,Y -133.4798,Z 175,A -90.1116,B 7.8927,C 0.3739,E1 7.8951,E2 181.6613} C_DIS
LIN {X -4.1198,Y -133.6411,Z 175,A -88.5426,B 7.8927,C 0.3737,E1 7.8995,E2 180.0903} C_DIS
LIN {X 0.9672,Y -133.7006,Z 175,A -86.8817,B 7.8923,C 0.3824,E1 7.9039,E2 178.4932} C_DIS
Enddeposition()
LIN {X 0.9672,Y -133.7006,Z 175,A -86.8817,B 7.8923,C 0.3824,E1 7.9039,E2 178.4932} C_DIS
Startdeposition()
$VEL.CP = VEL_PRINT
LIN {X -3.1181,Y -134.5758,Z 175,A -89.1766,B 7.8919,C 0.3966,E1 7.8976,E2 180.8918} C_DIS
LIN {X -6.4784,Y -134.4548,Z 175,A -90.3318,B 7.8922,C 0.3919,E1 7.8944,E2 182.0132} C_DIS
LIN {X -10.2741,Y -134.2186,Z 175,A -91.9121,B 7.8922,C 0.3912,E1 7.89,E2 183.5894} C_DIS
LIN {X -13.757,Y -133.9071,Z 175,A -93.941,B 7.8918,C 0.4,E1 7.8842,E2 185.686} C_DIS
LIN {X -18.3638,Y -133.3536,Z 175,A -95.3685,B 7.8922,C 0.3903,E1 7.8804,E2 187.0463} C_DIS
LIN {X -22.1169,Y -132.7809,Z 175,A -96.9792,B 7.8922,C 0.3897,E1 7.876,E2 188.6569} C_DIS
LIN {X -25.5891,Y -132.156,Z 175,A -98.4876,B 7.8923,C 0.3892,E1 7.8718,E2 190.1666} C_DIS
LIN {X -29.3806,Y -131.3661,Z 175,A -100.2837,B 7.8923,C 0.3908,E1 7.8669,E2 191.9815} C_DIS
LIN {X -33.0108,Y -130.4998,Z 175,A -101.7286,B 7.8923,C 0.3876,E1 7.863,E2 193.4089} C_DIS
LIN {X -36.6808,Y -129.5168,Z 175,A -103.3606,B 7.8924,C 0.3868,E1 7.8586,E2 195.0431} C_DIS
LIN {X -40.1646,Y -128.4805,Z 175,A -105.518,B 7.892,C 0.3955,E1 7.8527,E2 197.2763} C_DIS
LIN {X -44.7716,Y -126.9484,Z 175,A -107.0432,B 7.8925,C 0.3851,E1 7.8488,E2 198.735} C_DIS
LIN {X -49.0847,Y -125.3422,Z 175,A -108.98,B 7.8926,C 0.3829,E1 7.8438,E2 200.6693} C_DIS
LIN {X -52.1409,Y -124.1018,Z 175,A -110.4891,B 7.8926,C 0.3832,E1 7.8398,E2 202.1915} C_DIS
LIN {X -56.2261,Y -122.3051,Z 175,A -112.3209,B 7.8927,C 0.3801,E1 7.8352,E2 204.0151} C_DIS
LIN {X -59.2369,Y -120.8757,Z 175,A -113.7637,B 7.8928,C 0.3788,E1 7.8315,E2 205.4609} C_DIS
LIN {X -62.276,Y -119.3384,Z 175,A -115.1678,B 7.8929,C 0.3763,E1 7.8281,E2 206.8594} C_DIS
LIN {X -65.7924,Y -117.4384,Z 175,A -117.0049,B 7.8929,C 0.3763,E1 7.8235,E2 208.7133} C_DIS
LIN {X -69.8934,Y -115.0451,Z 175,A -118.9874,B 7.8931,C 0.3729,E1 7.8188,E2 210.691} C_DIS
LIN {X -73.5801,Y -112.7229,Z 175,A -120.9344,B 7.8931,C 0.3716,E1 7.8142,E2 212.6493} C_DIS
LIN {X -76.7543,Y -110.5856,Z 175,A -123.1218,B 7.8929,C 0.3776,E1 7.809,E2 214.9052} C_DIS
LIN {X -80.9644,Y -107.5415,Z 175,A -124.7496,B 7.8934,C 0.3652,E1 7.8055,E2 216.4609} C_DIS
LIN {X -85.5115,Y -103.9631,Z 175,A -127.3114,B 7.8936,C 0.3624,E1 7.7999,E2 219.0345} C_DIS
LIN {X -88.9326,Y -101.0517,Z 175,A -129.1783,B 7.8938,C 0.3583,E1 7.796,E2 220.8954} C_DIS
LIN {X -91.8047,Y -98.4494,Z 175,A -130.9065,B 7.8938,C 0.3564,E1 7.7924,E2 222.6328} C_DIS
LIN {X -95.1949,Y -95.176,Z 175,A -132.9466,B 7.894,C 0.353,E1 7.7883,E2 224.6766} C_DIS
LIN {X -97.4533,Y -92.8615,Z 175,A -134.3594,B 7.894,C 0.3507,E1 7.7856,E2 226.0935} C_DIS
LIN {X -100.3056,Y -89.7728,Z 175,A -136.1583,B 7.8943,C 0.3472,E1 7.7822,E2 227.8929} C_DIS
LIN {X -103.352,Y -86.2488,Z 175,A -138.115,B 7.8945,C 0.3426,E1 7.7787,E2 229.8457} C_DIS
LIN {X -105.3667,Y -83.775,Z 175,A -139.8912,B 7.8943,C 0.3456,E1 7.7755,E2 231.6725} C_DIS
LIN {X -107.9281,Y -80.4481,Z 175,A -141.2622,B 7.8947,C 0.3356,E1 7.7733,E2 232.9919} C_DIS
LIN {X -110.2609,Y -77.2207,Z 175,A -143.4371,B 7.8947,C 0.3386,E1 7.7697,E2 235.2248} C_DIS
LIN {X -112.6497,Y -73.6925,Z 175,A -144.9162,B 7.895,C 0.3296,E1 7.7675,E2 236.6622} C_DIS
LIN {X -114.978,Y -70.0043,Z 175,A -146.7989,B 7.8952,C 0.3255,E1 7.7647,E2 238.5471} C_DIS
LIN {X -118.4838,Y -63.8895,Z 175,A -150.0924,B 7.8953,C 0.3222,E1 7.7602,E2 241.8747} C_DIS
LIN {X -120.1193,Y -60.7561,Z 175,A -151.2892,B 7.8956,C 0.3141,E1 7.7587,E2 243.0332} C_DIS
LIN {X -122.5693,Y -55.6524,Z 175,A -153.7717,B 7.8958,C 0.3089,E1 7.7557,E2 245.5231} C_DIS
LIN {X -124.067,Y -52.2241,Z 175,A -155.3331,B 7.896,C 0.3043,E1 7.754,E2 247.0797} C_DIS
LIN {X -125.3685,Y -49.0171,Z 175,A -156.9129,B 7.896,C 0.3019,E1 7.7524,E2 248.6716} C_DIS
LIN {X -126.8919,Y -44.9321,Z 175,A -158.6992,B 7.8963,C 0.296,E1 7.7507,E2 250.4482} C_DIS
LIN {X -127.9447,Y -41.8397,Z 175,A -160.1099,B 7.8965,C 0.2925,E1 7.7494,E2 251.8604} C_DIS
LIN {X -129.7571,Y -35.8216,Z 175,A -162.7451,B 7.8967,C 0.2846,E1 7.7474,E2 254.4888} C_DIS
LIN {X -131.2468,Y -29.9027,Z 175,A -165.4745,B 7.8969,C 0.2792,E1 7.7455,E2 257.2324} C_DIS
LIN {X -132.0599,Y -26.0901,Z 175,A -167.2987,B 7.897,C 0.2768,E1 7.7445,E2 259.0754} C_DIS
LIN {X -132.747,Y -22.32,Z 175,A -168.883,B 7.8972,C 0.2715,E1 7.7437,E2 260.6527} C_DIS
LIN {X -133.3495,Y -18.3921,Z 175,A -170.6237,B 7.8973,C 0.2674,E1 7.743,E2 262.3981} C_DIS
LIN {X -133.8087,Y -14.6718,Z 175,A -172.2119,B 7.8975,C 0.2627,E1 7.7425,E2 263.9841} C_DIS
LIN {X -134.1774,Y -10.8016,Z 175,A -173.9999,B 7.8975,C 0.2598,E1 7.7421,E2 265.7869} C_DIS
LIN {X -134.4265,Y -7.0399,Z 175,A -175.5173,B 7.8978,C 0.254,E1 7.7418,E2 267.2922} C_DIS
LIN {X -134.5572,Y -3.7893,Z 175,A -176.9818,B 7.8978,C 0.2511,E1 7.7417,E2 268.7652} C_DIS
LIN {X -134.6108,Y 0.4701,Z 175,A -178.8786,B 7.898,C 0.247,E1 7.7417,E2 270.6706} C_DIS
LIN {X -134.5309,Y 4.6654,Z 175,A 179.3059,B 7.8981,C 0.2422,E1 7.7417,E2 272.4881} C_DIS
LIN {X -134.3332,Y 8.6428,Z 175,A 177.6812,B 7.8983,C 0.2364,E1 7.742,E2 274.1027} C_DIS
LIN {X -133.9999,Y 12.8057,Z 175,A 175.7951,B 7.8984,C 0.2328,E1 7.7425,E2 276.0003} C_DIS
LIN {X -133.5306,Y 17.0223,Z 175,A 173.9954,B 7.8986,C 0.2275,E1 7.7431,E2 277.7976} C_DIS
LIN {X -133.0394,Y 20.5052,Z 175,A 172.5496,B 7.8987,C 0.2225,E1 7.7437,E2 279.2357} C_DIS
LIN {X -132.5961,Y 23.2047,Z 175,A 171.2415,B 7.8987,C 0.2211,E1 7.7443,E2 280.5601} C_DIS
LIN {X -131.843,Y 27.1559,Z 175,A 169.5476,B 7.8989,C 0.216,E1 7.7452,E2 282.2501} C_DIS
LIN {X -130.9721,Y 31.0873,Z 175,A 167.8364,B 7.899,C 0.2112,E1 7.7463,E2 283.9594} C_DIS
LIN {X -130.1246,Y 34.4606,Z 175,A 166.2515,B 7.8991,C 0.2084,E1 7.7474,E2 285.5555} C_DIS
LIN {X -129.1457,Y 37.9642,Z 175,A 164.7405,B 7.8992,C 0.2036,E1 7.7485,E2 287.0604} C_DIS
LIN {X -128.0922,Y 41.3817,Z 175,A 163.0746,B 7.8992,C 0.2013,E1 7.75,E2 288.7422} C_DIS
LIN {X -127.1522,Y 44.1836,Z 175,A 161.2463,B 7.8992,C 0.2056,E1 7.7517,E2 290.6373} C_DIS
LIN {X -125.3813,Y 48.9841,Z 175,A 159.6839,B 7.8995,C 0.1914,E1 7.7532,E2 292.1242} C_DIS
LIN {X -123.8664,Y 52.7026,Z 175,A 157.831,B 7.8995,C 0.1888,E1 7.7552,E2 293.9926} C_DIS
LIN {X -122.3796,Y 56.065,Z 175,A 156.3221,B 7.8997,C 0.1839,E1 7.7569,E2 295.4933} C_DIS
LIN {X -121.0693,Y 58.8446,Z 175,A 155.0316,B 7.8997,C 0.1802,E1 7.7585,E2 296.7805} C_DIS
LIN {X -119.4633,Y 62.0381,Z 175,A 153.5721,B 7.8999,C 0.1754,E1 7.7603,E2 298.231} C_DIS
LIN {X -117.069,Y 66.4475,Z 175,A 151.3529,B 7.8999,C 0.1712,E1 7.7633,E2 300.4581} C_DIS
LIN {X -115.0871,Y 69.8237,Z 175,A 149.2946,B 7.8999,C 0.1724,E1 7.7663,E2 302.5616} C_DIS
LIN {X -113.3093,Y 72.6732,Z 175,A 148.108,B 7.9001,C 0.1655,E1 7.7681,E2 303.7179} C_DIS
LIN {X -110.6609,Y 76.6457,Z 175,A 145.9646,B 7.9001,C 0.1622,E1 7.7714,E2 305.8726} C_DIS
LIN {X -107.8744,Y 80.5203,Z 175,A 144.015,B 7.9003,C 0.1563,E1 7.7746,E2 307.8104} C_DIS
LIN {X -105.3715,Y 83.7689,Z 175,A 142.1544,B 7.9003,C 0.1539,E1 7.7778,E2 309.683} C_DIS
LIN {X -102.2144,Y 87.594,Z 175,A 139.9844,B 7.9004,C 0.15,E1 7.7817,E2 311.858} C_DIS
LIN {X -99.7834,Y 90.353,Z 175,A 138.2501,B 7.9004,C 0.149,E1 7.785,E2 313.611} C_DIS
LIN {X -97.6,Y 92.7081,Z 175,A 137.0145,B 7.9005,C 0.1443,E1 7.7874,E2 314.8297} C_DIS
LIN {X -94.87,Y 95.499,Z 175,A 135.2313,B 7.9005,C 0.1426,E1 7.7909,E2 316.6258} C_DIS
LIN {X -91.2006,Y 99.0093,Z 175,A 133.4327,B 7.9007,C 0.1331,E1 7.7945,E2 318.3792} C_DIS
LIN {X -87.8998,Y 101.951,Z 175,A 131.2658,B 7.9007,C 0.1336,E1 7.7991,E2 320.5783} C_DIS
LIN {X -84.713,Y 104.6143,Z 175,A 129.4533,B 7.9007,C 0.131,E1 7.803,E2 322.3945} C_DIS
LIN {X -81.4367,Y 107.185,Z 175,A 127.7798,B 7.9008,C 0.1264,E1 7.8067,E2 324.0547} C_DIS
LIN {X -78.5264,Y 109.3346,Z 175,A 125.8928,B 7.9008,C 0.1288,E1 7.811,E2 325.9815} C_DIS
LIN {X -75.7084,Y 111.3045,Z 175,A 124.6397,B 7.9008,C 0.1234,E1 7.8138,E2 327.2085} C_DIS
LIN {X -72.2714,Y 113.5665,Z 175,A 122.9979,B 7.9009,C 0.119,E1 7.8177,E2 328.8358} C_DIS
LIN {X -68.1133,Y 116.1076,Z 175,A 120.8264,B 7.9009,C 0.1173,E1 7.8229,E2 331.017} C_DIS
LIN {X -64.6084,Y 118.0939,Z 175,A 119.0856,B 7.9009,C 0.1153,E1 7.8271,E2 332.7596} C_DIS
LIN {X -58.9294,Y 121.0274,Z 175,A 116.2924,B 7.901,C 0.1128,E1 7.8341,E2 335.5593} C_DIS
LIN {X -55.188,Y 122.777,Z 175,A 114.6823,B 7.901,C 0.1084,E1 7.8381,E2 337.1503} C_DIS
LIN {X -52.157,Y 124.0951,Z 175,A 113.1458,B 7.901,C 0.1088,E1 7.8421,E2 338.7011} C_DIS
LIN {X -45.333,Y 126.7474,Z 175,A 109.7687,B 7.901,C 0.1096,E1 7.851,E2 342.107} C_DIS
LIN {X -42.1769,Y 127.8324,Z 175,A 108.6629,B 7.9012,C 0.1034,E1 7.8538,E2 343.1744} C_DIS
LIN {X -35.7551,Y 129.7757,Z 175,A 105.65,B 7.9012,C 0.1035,E1 7.862,E2 346.2041} C_DIS
LIN {X -31.8435,Y 130.7899,Z 175,A 104.0327,B 7.9012,C 0.1007,E1 7.8663,E2 347.8081} C_DIS
LIN {X -28.1762,Y 131.6285,Z 175,A 102.4232,B 7.9012,C 0.0998,E1 7.8707,E2 349.4176} C_DIS
LIN {X -24.2139,Y 132.4155,Z 175,A 100.6302,B 7.9012,C 0.1,E1 7.8756,E2 351.2183} C_DIS
LIN {X -20.5418,Y 133.0337,Z 175,A 99.1367,B 7.9012,C 0.0978,E1 7.8797,E2 352.7} C_DIS
LIN {X -16.7902,Y 133.561,Z 175,A 97.5036,B 7.9012,C 0.0975,E1 7.8842,E2 354.3347} C_DIS
LIN {X -13.3934,Y 133.9435,Z 175,A 95.9747,B 7.9012,C 0.0983,E1 7.8885,E2 355.8716} C_DIS
LIN {X -10.0749,Y 134.2332,Z 175,A 94.5574,B 7.9012,C 0.0979,E1 7.8925,E2 357.2881} C_DIS
LIN {X -5.59,Y 134.4948,Z 175,A 92.704,B 7.9012,C 0.0967,E1 7.8976,E2 359.1335} C_DIS
LIN {X -1.5859,Y 134.6028,Z 175,A 90.4556,B 7.9012,C 0.1055,E1 7.9041,E2 361.4455} C_DIS
LIN {X 3.0568,Y 134.5775,Z 175,A 88.9805,B 7.9012,C 0.0973,E1 7.908,E2 362.8605} C_DIS
LIN {X 6.9726,Y 134.4299,Z 175,A 87.3721,B 7.9012,C 0.0965,E1 7.9125,E2 364.4611} C_DIS
LIN {X 10.9423,Y 134.1655,Z 175,A 85.7017,B 7.9012,C 0.0965,E1 7.9171,E2 366.1281} C_DIS
LIN {X 15.5622,Y 133.7083,Z 175,A 83.6629,B 7.9012,C 0.0981,E1 7.9228,E2 368.1736} C_DIS
LIN {X 19.0265,Y 133.2589,Z 175,A 82.2237,B 7.9012,C 0.0979,E1 7.9268,E2 369.6067} C_DIS
LIN {X 22.9807,Y 132.6362,Z 175,A 80.4188,B 7.9012,C 0.1004,E1 7.9318,E2 371.4231} C_DIS
LIN {X 26.3042,Y 132.0163,Z 175,A 79.0137,B 7.9012,C 0.1006,E1 7.9356,E2 372.8238} C_DIS
LIN {X 30.0112,Y 131.2221,Z 175,A 77.4917,B 7.9012,C 0.1,E1 7.9397,E2 374.3344} C_DIS
LIN {X 33.5826,Y 130.3547,Z 175,A 75.9248,B 7.9012,C 0.1012,E1 7.944,E2 375.9013} C_DIS
LIN {X 37.129,Y 129.3897,Z 175,A 73.7836,B 7.901,C 0.1123,E1 7.9499,E2 378.1108} C_DIS
LIN {X 41.7724,Y 127.9671,Z 175,A 72.2237,B 7.9011,C 0.1054,E1 7.9539,E2 379.6102} C_DIS
LIN {X 46.1949,Y 126.4366,Z 175,A 70.2077,B 7.9011,C 0.1077,E1 7.9592,E2 381.6287} C_DIS
LIN {X 49.2913,Y 125.2618,Z 175,A 68.7949,B 7.9011,C 0.1092,E1 7.9629,E2 383.0418} C_DIS
LIN {X 53.0367,Y 123.722,Z 175,A 67.1859,B 7.9011,C 0.1091,E1 7.967,E2 384.6369} C_DIS
LIN {X 56.0189,Y 122.401,Z 175,A 65.7738,B 7.9011,C 0.1111,E1 7.9706,E2 386.0517} C_DIS
LIN {X 59.1621,Y 120.9126,Z 175,A 64.438,B 7.9011,C 0.1104,E1 7.9739,E2 387.3703} C_DIS
LIN {X 62.3262,Y 119.312,Z 175,A 62.8614,B 7.9011,C 0.1136,E1 7.9779,E2 388.9549} C_DIS
LIN {X 66.1541,Y 117.2351,Z 175,A 60.9316,B 7.901,C 0.1175,E1 7.9826,E2 390.8939} C_DIS
LIN {X 69.6947,Y 115.1652,Z 175,A 59.27,B 7.901,C 0.1185,E1 7.9866,E2 392.5456} C_DIS
LIN {X 73.1223,Y 113.0201,Z 175,A 57.505,B 7.9009,C 0.122,E1 7.9907,E2 394.316} C_DIS
LIN {X 77.8293,Y 109.8319,Z 175,A 55.1297,B 7.9009,C 0.1251,E1 7.9962,E2 396.6862} C_DIS
LIN {X 80.9618,Y 107.5434,Z 175,A 53.5301,B 7.9009,C 0.127,E1 7.9998,E2 398.2799} C_DIS
LIN {X 84.0754,Y 105.1276,Z 175,A 51.8285,B 7.9008,C 0.1304,E1 8.0035,E2 399.9847} C_DIS
LIN {X 87.5257,Y 102.2732,Z 175,A 49.9075,B 7.9008,C 0.1342,E1 8.0076,E2 401.9079} C_DIS
LIN {X 90.7836,Y 99.3926,Z 175,A 48.0806,B 7.9006,C 0.1373,E1 8.0114,E2 403.7324} C_DIS
LIN {X 94.0176,Y 96.3388,Z 175,A 46.2412,B 7.9006,C 0.14,E1 8.0151,E2 405.5658} C_DIS
LIN {X 97.1329,Y 93.1968,Z 175,A 44.3607,B 7.9006,C 0.1438,E1 8.0188,E2 407.4466} C_DIS
LIN {X 100.198,Y 89.8929,Z 175,A 42.5036,B 7.9005,C 0.1467,E1 8.0222,E2 409.297} C_DIS
LIN {X 103.0028,Y 86.6651,Z 175,A 40.6377,B 7.9004,C 0.1515,E1 8.0256,E2 411.1691} C_DIS
LIN {X 107.2066,Y 81.4082,Z 175,A 37.8407,B 7.9003,C 0.1567,E1 8.0305,E2 413.959} C_DIS
LIN {X 109.8554,Y 77.796,Z 175,A 35.9879,B 7.9003,C 0.1601,E1 8.0335,E2 415.8061} C_DIS
LIN {X 112.3553,Y 74.1397,Z 175,A 34.1354,B 7.9001,C 0.164,E1 8.0363,E2 417.6556} C_DIS
LIN {X 114.8616,Y 70.1943,Z 175,A 32.1812,B 7.9001,C 0.1681,E1 8.0392,E2 419.6065} C_DIS
LIN {X 116.9954,Y 66.5769,Z 175,A 30.4349,B 7.9,C 0.1718,E1 8.0417,E2 421.3487} C_DIS
LIN {X 119.0303,Y 62.8626,Z 175,A 28.7691,B 7.9,C 0.1736,E1 8.0439,E2 422.9989} C_DIS
LIN {X 120.5458,Y 59.9057,Z 175,A 27.3119,B 7.8998,C 0.1781,E1 8.0457,E2 424.4621} C_DIS
LIN {X 122.0039,Y 56.8777,Z 175,A 26.0282,B 7.8998,C 0.1789,E1 8.0472,E2 425.7288} C_DIS
LIN {X 123.4801,Y 53.5962,Z 175,A 24.4993,B 7.8998,C 0.1829,E1 8.049,E2 427.2583} C_DIS
LIN {X 124.6925,Y 50.7129,Z 175,A 23.2925,B 7.8998,C 0.184,E1 8.0502,E2 428.4508} C_DIS
LIN {X 126.8569,Y 45.0292,Z 175,A 20.4651,B 7.8994,C 0.1957,E1 8.053,E2 431.3092} C_DIS
LIN {X 128.318,Y 40.675,Z 175,A 18.581,B 7.8994,C 0.1996,E1 8.0547,E2 433.1859} C_DIS
LIN {X 129.5592,Y 36.5292,Z 175,A 16.7936,B 7.8992,C 0.2036,E1 8.0561,E2 434.968} C_DIS
LIN {X 130.5385,Y 32.8582,Z 175,A 15.2485,B 7.8992,C 0.2067,E1 8.0571,E2 436.5055} C_DIS
LIN {X 131.4982,Y 28.7797,Z 175,A 13.5021,B 7.899,C 0.2109,E1 8.0582,E2 438.2487} C_DIS
LIN {X 132.1563,Y 25.5876,Z 175,A 12.1626,B 7.899,C 0.2139,E1 8.0589,E2 439.5834} C_DIS
LIN {X 132.7707,Y 22.1779,Z 175,A 10.7255,B 7.8989,C 0.2173,E1 8.0596,E2 441.0171} C_DIS
LIN {X 133.2278,Y 19.2439,Z 175,A 9.4151,B 7.8987,C 0.2219,E1 8.0602,E2 442.3342} C_DIS
LIN {X 133.7315,Y 15.3679,Z 175,A 7.7841,B 7.8987,C 0.226,E1 8.0607,E2 443.9626} C_DIS
LIN {X 134.123,Y 11.4457,Z 175,A 6.1795,B 7.8985,C 0.2293,E1 8.0611,E2 445.5596} C_DIS
LIN {X 134.3909,Y 7.7063,Z 175,A 4.3632,B 7.8983,C 0.2383,E1 8.0615,E2 447.4042} C_DIS
LIN {X 134.5839,Y 2.7185,Z 175,A 2.506,B 7.8983,C 0.2391,E1 8.0616,E2 449.2306} C_DIS
LIN {X 134.607,Y -1.1133,Z 175,A 0.9361,B 7.8981,C 0.2426,E1 8.0616,E2 450.7944} C_DIS
LIN {X 134.5216,Y -4.9038,Z 175,A -0.6834,B 7.898,C 0.2474,E1 8.0615,E2 452.4161} C_DIS
LIN {X 134.1914,Y -10.6357,Z 175,A -3.1087,B 7.8978,C 0.2541,E1 8.0611,E2 454.8414} C_DIS
LIN {X 133.8298,Y -14.4757,Z 175,A -4.6826,B 7.8977,C 0.2574,E1 8.0606,E2 456.4084} C_DIS
LIN {X 133.3193,Y -18.604,Z 175,A -6.3963,B 7.8975,C 0.2614,E1 8.06,E2 458.1168} C_DIS
LIN {X 132.8665,Y -21.6037,Z 175,A -7.7233,B 7.8974,C 0.2658,E1 8.0594,E2 459.4493} C_DIS
LIN {X 132.3284,Y -24.6873,Z 175,A -8.9761,B 7.8974,C 0.268,E1 8.0588,E2 460.6937} C_DIS
LIN {X 131.6406,Y -28.1202,Z 175,A -10.4584,B 7.8972,C 0.2721,E1 8.058,E2 462.1764} C_DIS
LIN {X 130.828,Y -31.6852,Z 175,A -11.9279,B 7.8971,C 0.2747,E1 8.057,E2 463.6366} C_DIS
LIN {X 129.2127,Y -37.7355,Z 175,A -14.5451,B 7.8969,C 0.2813,E1 8.0551,E2 466.2505} C_DIS
LIN {X 128.3252,Y -40.6525,Z 175,A -15.8312,B 7.8967,C 0.2846,E1 8.0541,E2 467.5365} C_DIS
LIN {X 127.5133,Y -43.1351,Z 175,A -17.107,B 7.8965,C 0.291,E1 8.0529,E2 468.8336} C_DIS
LIN {X 126.169,Y -46.9185,Z 175,A -18.6305,B 7.8965,C 0.292,E1 8.0515,E2 470.3359} C_DIS
LIN {X 124.9989,Y -49.953,Z 175,A -20.057,B 7.8963,C 0.2966,E1 8.05,E2 471.769} C_DIS
LIN {X 123.6311,Y -53.2469,Z 175,A -21.4068,B 7.8963,C 0.2973,E1 8.0486,E2 473.0994} C_DIS
LIN {X 122.0443,Y -56.7902,Z 175,A -23.683,B 7.8956,C 0.3141,E1 8.0458,E2 475.4543} C_DIS
LIN {X 119.9677,Y -61.0538,Z 175,A -25.0722,B 7.8959,C 0.3069,E1 8.0442,E2 476.7678} C_DIS
LIN {X 118.5835,Y -63.7051,Z 175,A -26.8389,B 7.8954,C 0.32,E1 8.0418,E2 478.5969} C_DIS
LIN {X 116.4729,Y -67.4866,Z 175,A -28.1955,B 7.8956,C 0.3151,E1 8.04,E2 479.8952} C_DIS
LIN {X 114.2233,Y -71.228,Z 175,A -30.2467,B 7.8952,C 0.3236,E1 8.0369,E2 481.9722} C_DIS
LIN {X 111.4446,Y -75.5016,Z 175,A -32.4112,B 7.895,C 0.3288,E1 8.0336,E2 484.1382} C_DIS
LIN {X 109.5987,Y -78.1571,Z 175,A -33.5852,B 7.895,C 0.3281,E1 8.0317,E2 485.2885} C_DIS
LIN {X 107.6203,Y -80.8594,Z 175,A -35.0962,B 7.8948,C 0.3332,E1 8.0292,E2 486.8115} C_DIS
LIN {X 104.4769,Y -84.8829,Z 175,A -37.1554,B 7.8948,C 0.336,E1 8.0256,E2 488.8587} C_DIS
LIN {X 101.1442,Y -88.828,Z 175,A -39.297,B 7.8946,C 0.3399,E1 8.0217,E2 490.9955} C_DIS
LIN {X 98.2367,Y -92.033,Z 175,A -41.1401,B 7.8944,C 0.3439,E1 8.0182,E2 492.8405} C_DIS
LIN {X 95.1654,Y -95.2055,Z 175,A -42.9861,B 7.8942,C 0.3473,E1 8.0146,E2 494.6842} C_DIS
LIN {X 91.9588,Y -98.3058,Z 175,A -44.7715,B 7.8942,C 0.349,E1 8.011,E2 496.4573} C_DIS
LIN {X 89.6635,Y -100.4035,Z 175,A -46.0981,B 7.894,C 0.3518,E1 8.0083,E2 497.7855} C_DIS
LIN {X 86.5008,Y -103.1406,Z 175,A -47.8656,B 7.894,C 0.355,E1 8.0045,E2 499.5531} C_DIS
LIN {X 82.6818,Y -106.227,Z 175,A -50.1058,B 7.8936,C 0.3618,E1 7.9996,E2 501.8138} C_DIS
LIN {X 79.1905,Y -108.8545,Z 175,A -51.6352,B 7.8937,C 0.3589,E1 7.9962,E2 503.3038} C_DIS
LIN {X 76.6006,Y -110.6925,Z 175,A -53.1545,B 7.8935,C 0.3644,E1 7.9927,E2 504.8452} C_DIS
LIN {X 73.0378,Y -113.075,Z 175,A -54.9386,B 7.8934,C 0.3667,E1 7.9885,E2 506.626} C_DIS
LIN {X 69.9265,Y -115.025,Z 175,A -57.1293,B 7.8927,C 0.3809,E1 7.9831,E2 508.8959} C_DIS
LIN {X 65.0851,Y -117.8314,Z 175,A -59.0271,B 7.893,C 0.3755,E1 7.9786,E2 510.7358} C_DIS
LIN {X 61.0009,Y -119.9947,Z 175,A -60.7155,B 7.893,C 0.3732,E1 7.9745,E2 512.391} C_DIS
LIN {X 57.5842,Y -121.6722,Z 175,A -62.4234,B 7.8929,C 0.377,E1 7.9702,E2 514.1111} C_DIS
LIN {X 54.1264,Y -123.2508,Z 175,A -64.0198,B 7.8929,C 0.3787,E1 7.9661,E2 515.7063} C_DIS
LIN {X 50.4771,Y -124.7876,Z 175,A -65.5215,B 7.8929,C 0.3773,E1 7.9623,E2 517.1863} C_DIS
LIN {X 47.418,Y -125.9819,Z 175,A -67.0242,B 7.8927,C 0.3809,E1 7.9584,E2 518.7031} C_DIS
LIN {X 44.2592,Y -127.126,Z 175,A -68.3887,B 7.8927,C 0.3812,E1 7.9548,E2 520.0605} C_DIS
LIN {X 40.6832,Y -128.3154,Z 175,A -70.0389,B 7.8926,C 0.3836,E1 7.9504,E2 521.7176} C_DIS
LIN {X 36.5663,Y -129.5488,Z 175,A -71.8538,B 7.8926,C 0.3851,E1 7.9455,E2 523.5321} C_DIS
LIN {X 32.8873,Y -130.5311,Z 175,A -73.4436,B 7.8925,C 0.3859,E1 7.9412,E2 525.119} C_DIS
LIN {X 28.8139,Y -131.4908,Z 175,A -75.243,B 7.8924,C 0.3876,E1 7.9363,E2 526.9219} C_DIS
LIN {X 24.9908,Y -132.2704,Z 175,A -76.8102,B 7.8924,C 0.387,E1 7.9321,E2 528.4784} C_DIS
LIN {X 21.0544,Y -132.9544,Z 175,A -78.5512,B 7.8924,C 0.3887,E1 7.9272,E2 530.2256} C_DIS
LIN {X 17.795,Y -133.4293,Z 175,A -79.9632,B 7.8923,C 0.3896,E1 7.9233,E2 531.6396} C_DIS
LIN {X 14.3624,Y -133.842,Z 175,A -81.7515,B 7.892,C 0.3958,E1 7.9183,E2 533.4681} C_DIS
LIN {X 10.7168,Y -134.1845,Z 175,A -82.9729,B 7.8922,C 0.3905,E1 7.915,E2 534.6486} C_DIS
LIN {X 8.2759,Y -134.3558,Z 175,A -84.3573,B 7.8919,C 0.3968,E1 7.911,E2 536.0761} C_DIS
LIN {X 4.5375,Y -134.5357,Z 175,A -85.5959,B 7.8922,C 0.391,E1 7.9077,E2 537.2715} C_DIS
LIN {X 0.9786,Y -134.6055,Z 175,A -86.5038,B 7.8927,C 0.3808,E1 7.9053,E2 538.1039} C_DIS
Enddeposition()
LIN {X 0.9786,Y -134.6055,Z 175,A -86.5038,B 7.8927,C 0.3808,E1 7.9053,E2 538.1039} C_DIS
Startdeposition()
$VEL.CP = VEL_PRINT
LIN {X 2.8135,Y -135.489,Z 175,A -84.8568,B 7.711,C 0.3721,E1 7.7281,E2 536.4313} C_DIS
LIN {X 8.3422,Y -135.2599,Z 175,A -83.3438,B 7.7103,C 0.3858,E1 7.732,E2 535.0231} C_DIS
LIN {X 14.8747,Y -134.6986,Z 175,A -80.51,B 7.7104,C 0.3837,E1 7.7399,E2 532.18} C_DIS
LIN {X 18.382,Y -134.2666,Z 175,A -78.8317,B 7.7106,C 0.3798,E1 7.7446,E2 530.4774} C_DIS
LIN {X 22.2376,Y -133.6798,Z 175,A -77.3509,B 7.7106,C 0.3818,E1 7.7486,E2 529.017} C_DIS
LIN {X 25.8649,Y -133.0262,Z 175,A -75.8385,B 7.7106,C 0.3816,E1 7.7528,E2 527.5094} C_DIS
LIN {X 28.8287,Y -132.415,Z 175,A -74.5016,B 7.7106,C 0.3796,E1 7.7564,E2 526.1644} C_DIS
LIN {X 32.7899,Y -131.4911,Z 175,A -72.6977,B 7.7108,C 0.3768,E1 7.7614,E2 524.3487} C_DIS
LIN {X 36.9413,Y -130.3852,Z 175,A -71.0504,B 7.7108,C 0.3782,E1 7.7657,E2 522.7217} C_DIS
LIN {X 40.0439,Y -129.4658,Z 175,A -69.5338,B 7.7108,C 0.3742,E1 7.7698,E2 521.1852} C_DIS
LIN {X 44.3232,Y -128.0632,Z 175,A -67.7303,B 7.7109,C 0.3741,E1 7.7746,E2 519.393} C_DIS
LIN {X 47.7645,Y -126.8201,Z 175,A -66.1991,B 7.7109,C 0.3727,E1 7.7786,E2 517.8627} C_DIS
LIN {X 51.0599,Y -125.53,Z 175,A -64.7527,B 7.711,C 0.3718,E1 7.7823,E2 516.4216} C_DIS
LIN {X 54.0129,Y -124.2875,Z 175,A -63.386,B 7.7111,C 0.3699,E1 7.7859,E2 515.0522} C_DIS
LIN {X 57.4045,Y -122.759,Z 175,A -61.8797,B 7.7111,C 0.3691,E1 7.7897,E2 513.5531} C_DIS
LIN {X 60.0074,Y -121.5064,Z 175,A -60.6148,B 7.7113,C 0.3666,E1 7.7929,E2 512.2817} C_DIS
LIN {X 63.2776,Y -119.8363,Z 175,A -58.5741,B 7.7118,C 0.3553,E1 7.7981,E2 510.1773} C_DIS
LIN {X 67.287,Y -117.6339,Z 175,A -56.9228,B 7.7117,C 0.3576,E1 7.802,E2 508.5606} C_DIS
LIN {X 71.4481,Y -115.154,Z 175,A -55.1832,B 7.7116,C 0.3602,E1 7.806,E2 506.8587} C_DIS
LIN {X 74.7917,Y -113.0113,Z 175,A -53.3718,B 7.7118,C 0.3549,E1 7.8103,E2 505.029} C_DIS
LIN {X 78.8543,Y -110.2146,Z 175,A -51.3619,B 7.7119,C 0.3527,E1 7.8149,E2 503.0268} C_DIS
LIN {X 82.4069,Y -107.5842,Z 175,A -49.2627,B 7.7123,C 0.3449,E1 7.8196,E2 500.8966} C_DIS
LIN {X 85.0746,Y -105.4872,Z 175,A -48.2314,B 7.712,C 0.3499,E1 7.8218,E2 499.9153} C_DIS
LIN {X 87.9727,Y -103.083,Z 175,A -46.4338,B 7.7123,C 0.3428,E1 7.8257,E2 498.0901} C_DIS
LIN {X 91.2685,Y -100.1767,Z 175,A -44.7646,B 7.7123,C 0.3428,E1 7.8291,E2 496.4432} C_DIS
LIN {X 93.9498,Y -97.667,Z 175,A -43.1655,B 7.7125,C 0.3386,E1 7.8324,E2 494.8368} C_DIS
LIN {X 96.9163,Y -94.7234,Z 175,A -41.3875,B 7.7127,C 0.3347,E1 7.8359,E2 493.0556} C_DIS
LIN {X 99.8861,Y -91.5862,Z 175,A -39.5962,B 7.7128,C 0.3314,E1 7.8393,E2 491.267} C_DIS
LIN {X 102.7395,Y -88.3733,Z 175,A -37.6465,B 7.7131,C 0.3247,E1 7.8429,E2 489.2987} C_DIS
LIN {X 106.1544,Y -84.2409,Z 175,A -35.4649,B 7.7133,C 0.3212,E1 7.8467,E2 487.1257} C_DIS
LIN {X 108.5269,Y -81.1618,Z 175,A -33.9121,B 7.7133,C 0.3191,E1 7.8493,E2 485.5829} C_DIS
LIN {X 111.9578,Y -76.36,Z 175,A -31.5423,B 7.7135,C 0.3155,E1 7.8531,E2 483.2265} C_DIS
LIN {X 114.2676,Y -72.8568,Z 175,A -29.6166,B 7.7138,C 0.3081,E1 7.856,E2 481.2798} C_DIS
LIN {X 117.0143,Y -68.3593,Z 175,A -27.4519,B 7.714,C 0.3037,E1 7.8591,E2 479.1209} C_DIS
LIN {X 119.2344,Y -64.4088,Z 175,A -25.6693,B 7.714,C 0.3015,E1 7.8615,E2 477.3534} C_DIS
LIN {X 120.9365,Y -61.149,Z 175,A -24.1607,B 7.7142,C 0.2983,E1 7.8634,E2 475.849} C_DIS
LIN {X 124.2995,Y -53.9852,Z 175,A -21.1737,B 7.7142,C 0.2966,E1 7.8669,E2 472.9042} C_DIS
LIN {X 125.7471,Y -50.5215,Z 175,A -19.3614,B 7.7146,C 0.2878,E1 7.8688,E2 471.062} C_DIS
LIN {X 126.9606,Y -47.3893,Z 175,A -17.8372,B 7.7148,C 0.2819,E1 7.8703,E2 469.5233} C_DIS
LIN {X 128.5204,Y -42.9798,Z 175,A -16.0218,B 7.7148,C 0.2797,E1 7.872,E2 467.7264} C_DIS
LIN {X 129.5788,Y -39.6747,Z 175,A -14.5721,B 7.715,C 0.2759,E1 7.8732,E2 466.2774} C_DIS
LIN {X 130.597,Y -36.1841,Z 175,A -12.5086,B 7.7155,C 0.2611,E1 7.8748,E2 464.1458} C_DIS
LIN {X 131.8176,Y -31.4483,Z 175,A -11.1064,B 7.7153,C 0.2686,E1 7.8757,E2 462.8259} C_DIS
LIN {X 132.5022,Y -28.4247,Z 175,A -9.7839,B 7.7154,C 0.2646,E1 7.8764,E2 461.5007} C_DIS
LIN {X 133.1036,Y -25.4604,Z 175,A -8.5066,B 7.7155,C 0.261,E1 7.8771,E2 460.2223} C_DIS
LIN {X 133.6909,Y -22.1708,Z 175,A -7.1006,B 7.7157,C 0.2571,E1 7.8778,E2 458.816} C_DIS
LIN {X 134.315,Y -18.0129,Z 175,A -5.2916,B 7.7158,C 0.2514,E1 7.8785,E2 457.0013} C_DIS
LIN {X 134.7558,Y -14.3432,Z 175,A -3.8693,B 7.7159,C 0.2497,E1 7.8789,E2 455.5952} C_DIS
LIN {X 135.1128,Y -10.4757,Z 175,A -2.2373,B 7.716,C 0.2452,E1 7.8793,E2 453.9631} C_DIS
LIN {X 135.377,Y -6.1884,Z 175,A -0.3388,B 7.7163,C 0.2383,E1 7.8796,E2 452.0526} C_DIS
LIN {X 135.4931,Y -2.5666,Z 175,A 1.0645,B 7.7163,C 0.2365,E1 7.8797,E2 450.664} C_DIS
LIN {X 135.5139,Y 1.0488,Z 175,A 2.706,B 7.7165,C 0.2298,E1 7.8797,E2 449.007} C_DIS
LIN {X 135.4035,Y 5.5519,Z 175,A 4.3572,B 7.7165,C 0.2294,E1 7.8796,E2 447.386} C_DIS
LIN {X 135.2475,Y 8.5435,Z 175,A 5.6263,B 7.7166,C 0.2257,E1 7.8793,E2 446.1155} C_DIS
LIN {X 134.9728,Y 12.1549,Z 175,A 7.2817,B 7.7168,C 0.2188,E1 7.879,E2 444.4434} C_DIS
LIN {X 134.5597,Y 16.0779,Z 175,A 8.8213,B 7.7168,C 0.2166,E1 7.8785,E2 442.9183} C_DIS
LIN {X 134.1247,Y 19.3753,Z 175,A 10.1996,B 7.717,C 0.2131,E1 7.8779,E2 441.5424} C_DIS
LIN {X 133.4376,Y 23.6486,Z 175,A 11.9928,B 7.7171,C 0.2087,E1 7.8771,E2 439.7524} C_DIS
LIN {X 132.7997,Y 27.0006,Z 175,A 13.3766,B 7.7171,C 0.2058,E1 7.8764,E2 438.3749} C_DIS
LIN {X 132.1121,Y 30.1854,Z 175,A 14.7689,B 7.7173,C 0.2016,E1 7.8755,E2 436.9797} C_DIS
LIN {X 131.3102,Y 33.5026,Z 175,A 16.1265,B 7.7173,C 0.1993,E1 7.8746,E2 435.6316} C_DIS
LIN {X 130.4504,Y 36.7081,Z 175,A 17.555,B 7.7175,C 0.1949,E1 7.8736,E2 434.1989} C_DIS
LIN {X 129.0331,Y 41.4155,Z 175,A 19.5807,B 7.7175,C 0.1902,E1 7.8719,E2 432.1784} C_DIS
LIN {X 127.7962,Y 45.0934,Z 175,A 21.3702,B 7.7178,C 0.1829,E1 7.8702,E2 430.3694} C_DIS
LIN {X 125.8813,Y 50.1884,Z 175,A 23.3208,B 7.7178,C 0.1836,E1 7.8683,E2 428.4608} C_DIS
LIN {X 124.2492,Y 54.1014,Z 175,A 25.2264,B 7.7179,C 0.1766,E1 7.8662,E2 426.54} C_DIS
LIN {X 122.9792,Y 56.9283,Z 175,A 26.5322,B 7.7179,C 0.1733,E1 7.8647,E2 425.234} C_DIS
LIN {X 121.3965,Y 60.2303,Z 175,A 28.0517,B 7.7181,C 0.1699,E1 7.8629,E2 423.7171} C_DIS
LIN {X 119.3352,Y 64.2213,Z 175,A 29.9686,B 7.7181,C 0.1647,E1 7.8604,E2 421.7971} C_DIS
LIN {X 117.0926,Y 68.2256,Z 175,A 31.8938,B 7.7183,C 0.1602,E1 7.8577,E2 419.8728} C_DIS
LIN {X 114.7614,Y 72.0774,Z 175,A 33.793,B 7.7183,C 0.1556,E1 7.8549,E2 417.9732} C_DIS
LIN {X 112.2947,Y 75.8628,Z 175,A 35.6482,B 7.7184,C 0.1521,E1 7.852,E2 416.1239} C_DIS
LIN {X 109.6291,Y 79.6664,Z 175,A 37.5696,B 7.7184,C 0.1484,E1 7.8489,E2 414.2069} C_DIS
LIN {X 107.0432,Y 83.1084,Z 175,A 39.7944,B 7.7187,C 0.1365,E1 7.8451,E2 411.9311} C_DIS
LIN {X 104.214,Y 86.6299,Z 175,A 41.135,B 7.7186,C 0.1431,E1 7.8428,E2 410.6603} C_DIS
LIN {X 101.7711,Y 89.4875,Z 175,A 42.8539,B 7.7187,C 0.1373,E1 7.8396,E2 408.925} C_DIS
LIN {X 98.66,Y 92.9056,Z 175,A 44.7282,B 7.7187,C 0.1347,E1 7.8361,E2 407.0599} C_DIS
LIN {X 95.6176,Y 96.034,Z 175,A 46.5785,B 7.7188,C 0.1308,E1 7.8324,E2 405.2083} C_DIS
LIN {X 92.3875,Y 99.1453,Z 175,A 48.4333,B 7.7188,C 0.1278,E1 7.8287,E2 403.3582} C_DIS
LIN {X 88.9461,Y 102.2442,Z 175,A 50.3644,B 7.7189,C 0.1246,E1 7.8247,E2 401.4298} C_DIS
LIN {X 85.4851,Y 105.1555,Z 175,A 52.2647,B 7.7189,C 0.1214,E1 7.8206,E2 399.5306} C_DIS
LIN {X 82.1078,Y 107.8129,Z 175,A 54.0611,B 7.719,C 0.1186,E1 7.8166,E2 397.7365} C_DIS
LIN {X 78.4668,Y 110.4916,Z 175,A 55.9284,B 7.719,C 0.1162,E1 7.8124,E2 395.8743} C_DIS
LIN {X 73.7208,Y 113.7123,Z 175,A 58.291,B 7.719,C 0.1134,E1 7.8069,E2 393.5191} C_DIS
LIN {X 70.4463,Y 115.7701,Z 175,A 59.998,B 7.7191,C 0.1097,E1 7.8028,E2 391.8032} C_DIS
LIN {X 66.5249,Y 118.0666,Z 175,A 61.8816,B 7.7191,C 0.1076,E1 7.7983,E2 389.9242} C_DIS
LIN {X 62.521,Y 120.2336,Z 175,A 63.644,B 7.7191,C 0.1079,E1 7.794,E2 388.1815} C_DIS
LIN {X 59.3883,Y 121.8118,Z 175,A 65.1569,B 7.7191,C 0.1055,E1 7.7902,E2 386.665} C_DIS
LIN {X 56.2341,Y 123.3002,Z 175,A 66.6064,B 7.7192,C 0.1042,E1 7.7865,E2 385.2187} C_DIS
LIN {X 52.6749,Y 124.8611,Z 175,A 68.3294,B 7.7192,C 0.1009,E1 7.7821,E2 383.4861} C_DIS
LIN {X 48.7917,Y 126.4286,Z 175,A 70.0802,B 7.7192,C 0.0994,E1 7.7776,E2 381.7378} C_DIS
LIN {X 45.5304,Y 127.6398,Z 175,A 71.4733,B 7.7192,C 0.0994,E1 7.7739,E2 380.3545} C_DIS
LIN {X 42.5346,Y 128.6687,Z 175,A 72.8087,B 7.7192,C 0.0982,E1 7.7704,E2 379.0197} C_DIS
LIN {X 36.1536,Y 130.6055,Z 175,A 75.5529,B 7.7193,C 0.0972,E1 7.7631,E2 376.2853} C_DIS
LIN {X 33.0307,Y 131.43,Z 175,A 76.9009,B 7.7193,C 0.0965,E1 7.7594,E2 374.9397} C_DIS
LIN {X 29.9718,Y 132.1609,Z 175,A 78.3395,B 7.7193,C 0.0938,E1 7.7555,E2 373.4882} C_DIS
LIN {X 25.8649,Y 133.0262,Z 175,A 80.0945,B 7.7193,C 0.0931,E1 7.7507,E2 371.7361} C_DIS
LIN {X 22.3533,Y 133.6605,Z 175,A 81.5295,B 7.7193,C 0.0936,E1 7.7468,E2 370.3104} C_DIS
LIN {X 19.077,Y 134.1674,Z 175,A 82.9496,B 7.7193,C 0.0927,E1 7.7428,E2 368.8885} C_DIS
LIN {X 15.5383,Y 134.6241,Z 175,A 84.6588,B 7.7194,C 0.0889,E1 7.738,E2 367.1555} C_DIS
LIN {X 11.2794,Y 135.0467,Z 175,A 86.2357,B 7.7194,C 0.0923,E1 7.7337,E2 365.6076} C_DIS
LIN {X 7.8655,Y 135.2893,Z 175,A 87.7301,B 7.7194,C 0.0912,E1 7.7295,E2 364.108} C_DIS
LIN {X 3.8088,Y 135.4635,Z 175,A 89.3473,B 7.7194,C 0.0927,E1 7.7251,E2 362.5035} C_DIS
LIN {X -1.5642,Y 135.5097,Z 175,A 91.6405,B 7.7194,C 0.0923,E1 7.7187,E2 360.2089} C_DIS
LIN {X -4.9959,Y 135.4252,Z 175,A 93.2261,B 7.7194,C 0.0903,E1 7.7142,E2 358.6076} C_DIS
LIN {X -8.7356,Y 135.2357,Z 175,A 94.8514,B 7.7194,C 0.0899,E1 7.7096,E2 356.978} C_DIS
LIN {X -12.7785,Y 134.9132,Z 175,A 96.4823,B 7.7194,C 0.0917,E1 7.7051,E2 355.3582} C_DIS
LIN {X -16.0851,Y 134.5589,Z 175,A 97.8285,B 7.7194,C 0.0931,E1 7.7014,E2 354.02} C_DIS
LIN {X -19.2302,Y 134.1455,Z 175,A 99.2436,B 7.7194,C 0.0924,E1 7.6975,E2 352.5966} C_DIS
LIN {X -22.7811,Y 133.5891,Z 175,A 100.7008,B 7.7194,C 0.0941,E1 7.6935,E2 351.148} C_DIS
LIN {X -25.7403,Y 133.05,Z 175,A 101.9494,B 7.7194,C 0.0952,E1 7.6901,E2 349.9029} C_DIS
LIN {X -28.6695,Y 132.4494,Z 175,A 103.2554,B 7.7194,C 0.0952,E1 7.6865,E2 348.5926} C_DIS
LIN {X -31.7871,Y 131.7359,Z 175,A 104.7054,B 7.7194,C 0.0946,E1 7.6825,E2 347.1316} C_DIS
LIN {X -35.2981,Y 130.8394,Z 175,A 106.6564,B 7.7194,C 0.0893,E1 7.6771,E2 345.1306} C_DIS
LIN {X -39.3484,Y 129.6787,Z 175,A 107.7693,B 7.7193,C 0.1011,E1 7.6744,E2 344.1002} C_DIS
LIN {X -43.4737,Y 128.356,Z 175,A 109.8899,B 7.7193,C 0.0983,E1 7.6686,E2 341.946} C_DIS
LIN {X -51.2527,Y 125.4523,Z 175,A 113.3234,B 7.7193,C 0.1031,E1 7.6597,E2 338.5245} C_DIS
LIN {X -54.0175,Y 124.2855,Z 175,A 114.6251,B 7.7193,C 0.1041,E1 7.6564,E2 337.2197} C_DIS
LIN {X -57.0129,Y 122.94,Z 175,A 116.0469,B 7.7193,C 0.1052,E1 7.6527,E2 335.7949} C_DIS
LIN {X -63.3653,Y 119.7902,Z 175,A 118.9626,B 7.7191,C 0.1104,E1 7.6455,E2 332.8917} C_DIS
LIN {X -66.7469,Y 117.9415,Z 175,A 121.3563,B 7.7193,C 0.1013,E1 7.6395,E2 330.4062} C_DIS
LIN {X -71.2154,Y 115.2986,Z 175,A 122.8822,B 7.7191,C 0.1146,E1 7.636,E2 328.9639} C_DIS
LIN {X -74.2803,Y 113.3479,Z 175,A 124.5794,B 7.7191,C 0.1146,E1 7.632,E2 327.2483} C_DIS
LIN {X -78.2822,Y 110.6215,Z 175,A 126.7155,B 7.7191,C 0.1167,E1 7.6271,E2 325.1032} C_DIS
LIN {X -82.1753,Y 107.7613,Z 175,A 128.7146,B 7.719,C 0.1209,E1 7.6226,E2 323.1112} C_DIS
LIN {X -84.9974,Y 105.5495,Z 175,A 130.2214,B 7.719,C 0.1238,E1 7.6193,E2 321.6069} C_DIS
LIN {X -88.3196,Y 102.7858,Z 175,A 132.5898,B 7.719,C 0.1194,E1 7.6142,E2 319.1739} C_DIS
LIN {X -91.971,Y 99.5324,Z 175,A 133.8493,B 7.7187,C 0.135,E1 7.6118,E2 318.015} C_DIS
LIN {X -95.0115,Y 96.6337,Z 175,A 135.9385,B 7.7187,C 0.1342,E1 7.6075,E2 315.8894} C_DIS
LIN {X -98.1249,Y 93.4709,Z 175,A 138.0988,B 7.7187,C 0.134,E1 7.6033,E2 313.6962} C_DIS
LIN {X -100.4,Y 91.0224,Z 175,A 139.1003,B 7.7187,C 0.1429,E1 7.6015,E2 312.7463} C_DIS
LIN {X -102.4938,Y 88.6586,Z 175,A 140.6976,B 7.7187,C 0.1421,E1 7.5985,E2 311.1183} C_DIS
LIN {X -105.0608,Y 85.6009,Z 175,A 142.3548,B 7.7185,C 0.1463,E1 7.5955,E2 309.4665} C_DIS
Enddeposition()
END
